  gc_ErrTranslation_en_Texts : ARRAY[0..1193] OF POINTER TO WSTRING(101) := [ADR(gc_ErrTranslation_en_Text0), ADR(gc_ErrTranslation_en_Text1), ADR(gc_ErrTranslation_en_Text2), ADR(gc_ErrTranslation_en_Text3), ADR(gc_ErrTranslation_en_Text4), ADR(gc_ErrTranslation_en_Text5), ADR(gc_ErrTranslation_en_Text6), ADR(gc_ErrTranslation_en_Text7), ADR(gc_ErrTranslation_en_Text8), ADR(gc_ErrTranslation_en_Text9), ADR(gc_ErrTranslation_en_Text10), ADR(gc_ErrTranslation_en_Text11), ADR(gc_ErrTranslation_en_Text12), ADR(gc_ErrTranslation_en_Text13), ADR(gc_ErrTranslation_en_Text14), ADR(gc_ErrTranslation_en_Text15), ADR(gc_ErrTranslation_en_Text16), ADR(gc_ErrTranslation_en_Text17), ADR(gc_ErrTranslation_en_Text18), ADR(gc_ErrTranslation_en_Text19), ADR(gc_ErrTranslation_en_Text20), ADR(gc_ErrTranslation_en_Text21), ADR(gc_ErrTranslation_en_Text22), ADR(gc_ErrTranslation_en_Text23), ADR(gc_ErrTranslation_en_Text24), ADR(gc_ErrTranslation_en_Text25), ADR(gc_ErrTranslation_en_Text26), ADR(gc_ErrTranslation_en_Text27), ADR(gc_ErrTranslation_en_Text28), ADR(gc_ErrTranslation_en_Text29), ADR(gc_ErrTranslation_en_Text30), ADR(gc_ErrTranslation_en_Text31), ADR(gc_ErrTranslation_en_Text32), ADR(gc_ErrTranslation_en_Text33), ADR(gc_ErrTranslation_en_Text34), ADR(gc_ErrTranslation_en_Text35), ADR(gc_ErrTranslation_en_Text36), ADR(gc_ErrTranslation_en_Text37), ADR(gc_ErrTranslation_en_Text38), ADR(gc_ErrTranslation_en_Text39), ADR(gc_ErrTranslation_en_Text40), ADR(gc_ErrTranslation_en_Text41), ADR(gc_ErrTranslation_en_Text42), ADR(gc_ErrTranslation_en_Text43), ADR(gc_ErrTranslation_en_Text44), ADR(gc_ErrTranslation_en_Text45), ADR(gc_ErrTranslation_en_Text46), ADR(gc_ErrTranslation_en_Text47), ADR(gc_ErrTranslation_en_Text48), ADR(gc_ErrTranslation_en_Text49), ADR(gc_ErrTranslation_en_Text50), ADR(gc_ErrTranslation_en_Text51), ADR(gc_ErrTranslation_en_Text52), ADR(gc_ErrTranslation_en_Text53), ADR(gc_ErrTranslation_en_Text54), ADR(gc_ErrTranslation_en_Text55), ADR(gc_ErrTranslation_en_Text56), ADR(gc_ErrTranslation_en_Text57), ADR(gc_ErrTranslation_en_Text58), ADR(gc_ErrTranslation_en_Text59), ADR(gc_ErrTranslation_en_Text60), ADR(gc_ErrTranslation_en_Text61), ADR(gc_ErrTranslation_en_Text62), ADR(gc_ErrTranslation_en_Text63), ADR(gc_ErrTranslation_en_Text64), ADR(gc_ErrTranslation_en_Text65), ADR(gc_ErrTranslation_en_Text66), ADR(gc_ErrTranslation_en_Text67), ADR(gc_ErrTranslation_en_Text68), ADR(gc_ErrTranslation_en_Text69), ADR(gc_ErrTranslation_en_Text70), ADR(gc_ErrTranslation_en_Text71), ADR(gc_ErrTranslation_en_Text72), ADR(gc_ErrTranslation_en_Text73), ADR(gc_ErrTranslation_en_Text74), ADR(gc_ErrTranslation_en_Text75), ADR(gc_ErrTranslation_en_Text76), ADR(gc_ErrTranslation_en_Text77), ADR(gc_ErrTranslation_en_Text78), ADR(gc_ErrTranslation_en_Text79), ADR(gc_ErrTranslation_en_Text80), ADR(gc_ErrTranslation_en_Text81), ADR(gc_ErrTranslation_en_Text82), ADR(gc_ErrTranslation_en_Text83), ADR(gc_ErrTranslation_en_Text84), ADR(gc_ErrTranslation_en_Text85), ADR(gc_ErrTranslation_en_Text86), ADR(gc_ErrTranslation_en_Text87), ADR(gc_ErrTranslation_en_Text88), ADR(gc_ErrTranslation_en_Text89), ADR(gc_ErrTranslation_en_Text90), ADR(gc_ErrTranslation_en_Text91), ADR(gc_ErrTranslation_en_Text92), ADR(gc_ErrTranslation_en_Text93), ADR(gc_ErrTranslation_en_Text94), ADR(gc_ErrTranslation_en_Text95), ADR(gc_ErrTranslation_en_Text96), ADR(gc_ErrTranslation_en_Text97), ADR(gc_ErrTranslation_en_Text98), ADR(gc_ErrTranslation_en_Text99), ADR(gc_ErrTranslation_en_Text100), ADR(gc_ErrTranslation_en_Text101), ADR(gc_ErrTranslation_en_Text102), ADR(gc_ErrTranslation_en_Text103), ADR(gc_ErrTranslation_en_Text104), ADR(gc_ErrTranslation_en_Text105), ADR(gc_ErrTranslation_en_Text106), ADR(gc_ErrTranslation_en_Text107), ADR(gc_ErrTranslation_en_Text108), ADR(gc_ErrTranslation_en_Text109), ADR(gc_ErrTranslation_en_Text110), ADR(gc_ErrTranslation_en_Text111), ADR(gc_ErrTranslation_en_Text112), ADR(gc_ErrTranslation_en_Text113), ADR(gc_ErrTranslation_en_Text114), ADR(gc_ErrTranslation_en_Text115), ADR(gc_ErrTranslation_en_Text116), ADR(gc_ErrTranslation_en_Text117), ADR(gc_ErrTranslation_en_Text118), ADR(gc_ErrTranslation_en_Text119), ADR(gc_ErrTranslation_en_Text120), ADR(gc_ErrTranslation_en_Text121), ADR(gc_ErrTranslation_en_Text122), ADR(gc_ErrTranslation_en_Text123), ADR(gc_ErrTranslation_en_Text124), ADR(gc_ErrTranslation_en_Text125), ADR(gc_ErrTranslation_en_Text126), ADR(gc_ErrTranslation_en_Text127), ADR(gc_ErrTranslation_en_Text128), ADR(gc_ErrTranslation_en_Text129), ADR(gc_ErrTranslation_en_Text130), ADR(gc_ErrTranslation_en_Text131), ADR(gc_ErrTranslation_en_Text132), ADR(gc_ErrTranslation_en_Text133), ADR(gc_ErrTranslation_en_Text134), ADR(gc_ErrTranslation_en_Text135), ADR(gc_ErrTranslation_en_Text136), ADR(gc_ErrTranslation_en_Text137), ADR(gc_ErrTranslation_en_Text138), ADR(gc_ErrTranslation_en_Text139), ADR(gc_ErrTranslation_en_Text140), ADR(gc_ErrTranslation_en_Text141), ADR(gc_ErrTranslation_en_Text142), ADR(gc_ErrTranslation_en_Text143), ADR(gc_ErrTranslation_en_Text144), ADR(gc_ErrTranslation_en_Text145), ADR(gc_ErrTranslation_en_Text146), ADR(gc_ErrTranslation_en_Text147), ADR(gc_ErrTranslation_en_Text148), ADR(gc_ErrTranslation_en_Text149), ADR(gc_ErrTranslation_en_Text150), ADR(gc_ErrTranslation_en_Text151), ADR(gc_ErrTranslation_en_Text152), ADR(gc_ErrTranslation_en_Text153), ADR(gc_ErrTranslation_en_Text154), ADR(gc_ErrTranslation_en_Text155), ADR(gc_ErrTranslation_en_Text156), ADR(gc_ErrTranslation_en_Text157), ADR(gc_ErrTranslation_en_Text158), ADR(gc_ErrTranslation_en_Text159), ADR(gc_ErrTranslation_en_Text160), ADR(gc_ErrTranslation_en_Text161), ADR(gc_ErrTranslation_en_Text162), ADR(gc_ErrTranslation_en_Text163), ADR(gc_ErrTranslation_en_Text164), ADR(gc_ErrTranslation_en_Text165), ADR(gc_ErrTranslation_en_Text166), ADR(gc_ErrTranslation_en_Text167), ADR(gc_ErrTranslation_en_Text168), ADR(gc_ErrTranslation_en_Text169), ADR(gc_ErrTranslation_en_Text170), ADR(gc_ErrTranslation_en_Text171), ADR(gc_ErrTranslation_en_Text172), ADR(gc_ErrTranslation_en_Text173), ADR(gc_ErrTranslation_en_Text174), ADR(gc_ErrTranslation_en_Text175), ADR(gc_ErrTranslation_en_Text176), ADR(gc_ErrTranslation_en_Text177), ADR(gc_ErrTranslation_en_Text178), ADR(gc_ErrTranslation_en_Text179), ADR(gc_ErrTranslation_en_Text180), ADR(gc_ErrTranslation_en_Text181), ADR(gc_ErrTranslation_en_Text182), ADR(gc_ErrTranslation_en_Text183), ADR(gc_ErrTranslation_en_Text184), ADR(gc_ErrTranslation_en_Text185), ADR(gc_ErrTranslation_en_Text186), ADR(gc_ErrTranslation_en_Text187), ADR(gc_ErrTranslation_en_Text188), ADR(gc_ErrTranslation_en_Text189), ADR(gc_ErrTranslation_en_Text190), ADR(gc_ErrTranslation_en_Text191), ADR(gc_ErrTranslation_en_Text192), ADR(gc_ErrTranslation_en_Text193), ADR(gc_ErrTranslation_en_Text194), ADR(gc_ErrTranslation_en_Text195), ADR(gc_ErrTranslation_en_Text196), ADR(gc_ErrTranslation_en_Text197), ADR(gc_ErrTranslation_en_Text198), ADR(gc_ErrTranslation_en_Text199), ADR(gc_ErrTranslation_en_Text200), ADR(gc_ErrTranslation_en_Text201), ADR(gc_ErrTranslation_en_Text202), ADR(gc_ErrTranslation_en_Text203), ADR(gc_ErrTranslation_en_Text204), ADR(gc_ErrTranslation_en_Text205), ADR(gc_ErrTranslation_en_Text206), ADR(gc_ErrTranslation_en_Text207), ADR(gc_ErrTranslation_en_Text208), ADR(gc_ErrTranslation_en_Text209), ADR(gc_ErrTranslation_en_Text210), ADR(gc_ErrTranslation_en_Text211), ADR(gc_ErrTranslation_en_Text212), ADR(gc_ErrTranslation_en_Text213), ADR(gc_ErrTranslation_en_Text214), ADR(gc_ErrTranslation_en_Text215), ADR(gc_ErrTranslation_en_Text216), ADR(gc_ErrTranslation_en_Text217), ADR(gc_ErrTranslation_en_Text218), ADR(gc_ErrTranslation_en_Text219), ADR(gc_ErrTranslation_en_Text220), ADR(gc_ErrTranslation_en_Text221), ADR(gc_ErrTranslation_en_Text222), ADR(gc_ErrTranslation_en_Text223), ADR(gc_ErrTranslation_en_Text224), ADR(gc_ErrTranslation_en_Text225), ADR(gc_ErrTranslation_en_Text226), ADR(gc_ErrTranslation_en_Text227), ADR(gc_ErrTranslation_en_Text228), ADR(gc_ErrTranslation_en_Text229), ADR(gc_ErrTranslation_en_Text230), ADR(gc_ErrTranslation_en_Text231), ADR(gc_ErrTranslation_en_Text232), ADR(gc_ErrTranslation_en_Text233), ADR(gc_ErrTranslation_en_Text234), ADR(gc_ErrTranslation_en_Text235), ADR(gc_ErrTranslation_en_Text236), ADR(gc_ErrTranslation_en_Text237), ADR(gc_ErrTranslation_en_Text238), ADR(gc_ErrTranslation_en_Text239), ADR(gc_ErrTranslation_en_Text240), ADR(gc_ErrTranslation_en_Text241), ADR(gc_ErrTranslation_en_Text242), ADR(gc_ErrTranslation_en_Text243), ADR(gc_ErrTranslation_en_Text244), ADR(gc_ErrTranslation_en_Text245), ADR(gc_ErrTranslation_en_Text246), ADR(gc_ErrTranslation_en_Text247), ADR(gc_ErrTranslation_en_Text248), ADR(gc_ErrTranslation_en_Text249), ADR(gc_ErrTranslation_en_Text250), ADR(gc_ErrTranslation_en_Text251), ADR(gc_ErrTranslation_en_Text252), ADR(gc_ErrTranslation_en_Text253), ADR(gc_ErrTranslation_en_Text254), ADR(gc_ErrTranslation_en_Text255), ADR(gc_ErrTranslation_en_Text256), ADR(gc_ErrTranslation_en_Text257), ADR(gc_ErrTranslation_en_Text258), ADR(gc_ErrTranslation_en_Text259), ADR(gc_ErrTranslation_en_Text260), ADR(gc_ErrTranslation_en_Text261), ADR(gc_ErrTranslation_en_Text262), ADR(gc_ErrTranslation_en_Text263), ADR(gc_ErrTranslation_en_Text264), ADR(gc_ErrTranslation_en_Text265), ADR(gc_ErrTranslation_en_Text266), ADR(gc_ErrTranslation_en_Text267), ADR(gc_ErrTranslation_en_Text268), ADR(gc_ErrTranslation_en_Text269), ADR(gc_ErrTranslation_en_Text270), ADR(gc_ErrTranslation_en_Text271), ADR(gc_ErrTranslation_en_Text272), ADR(gc_ErrTranslation_en_Text273), ADR(gc_ErrTranslation_en_Text274), ADR(gc_ErrTranslation_en_Text275), ADR(gc_ErrTranslation_en_Text276), ADR(gc_ErrTranslation_en_Text277), ADR(gc_ErrTranslation_en_Text278), ADR(gc_ErrTranslation_en_Text279), ADR(gc_ErrTranslation_en_Text280), ADR(gc_ErrTranslation_en_Text281), ADR(gc_ErrTranslation_en_Text282), ADR(gc_ErrTranslation_en_Text283), ADR(gc_ErrTranslation_en_Text284), ADR(gc_ErrTranslation_en_Text285), ADR(gc_ErrTranslation_en_Text286), ADR(gc_ErrTranslation_en_Text287), ADR(gc_ErrTranslation_en_Text288), ADR(gc_ErrTranslation_en_Text289), ADR(gc_ErrTranslation_en_Text290), ADR(gc_ErrTranslation_en_Text291), ADR(gc_ErrTranslation_en_Text292), ADR(gc_ErrTranslation_en_Text293), ADR(gc_ErrTranslation_en_Text294), ADR(gc_ErrTranslation_en_Text295), ADR(gc_ErrTranslation_en_Text296), ADR(gc_ErrTranslation_en_Text297), ADR(gc_ErrTranslation_en_Text298), ADR(gc_ErrTranslation_en_Text299), ADR(gc_ErrTranslation_en_Text300), ADR(gc_ErrTranslation_en_Text301), ADR(gc_ErrTranslation_en_Text302), ADR(gc_ErrTranslation_en_Text303), ADR(gc_ErrTranslation_en_Text304), ADR(gc_ErrTranslation_en_Text305), ADR(gc_ErrTranslation_en_Text306), ADR(gc_ErrTranslation_en_Text307), ADR(gc_ErrTranslation_en_Text308), ADR(gc_ErrTranslation_en_Text309), ADR(gc_ErrTranslation_en_Text310), ADR(gc_ErrTranslation_en_Text311), ADR(gc_ErrTranslation_en_Text312), ADR(gc_ErrTranslation_en_Text313), ADR(gc_ErrTranslation_en_Text314), ADR(gc_ErrTranslation_en_Text315), ADR(gc_ErrTranslation_en_Text316), ADR(gc_ErrTranslation_en_Text317), ADR(gc_ErrTranslation_en_Text318), ADR(gc_ErrTranslation_en_Text319), ADR(gc_ErrTranslation_en_Text320), ADR(gc_ErrTranslation_en_Text321), ADR(gc_ErrTranslation_en_Text322), ADR(gc_ErrTranslation_en_Text323), ADR(gc_ErrTranslation_en_Text324), ADR(gc_ErrTranslation_en_Text325), ADR(gc_ErrTranslation_en_Text326), ADR(gc_ErrTranslation_en_Text327), ADR(gc_ErrTranslation_en_Text328), ADR(gc_ErrTranslation_en_Text329), ADR(gc_ErrTranslation_en_Text330), ADR(gc_ErrTranslation_en_Text331), ADR(gc_ErrTranslation_en_Text332), ADR(gc_ErrTranslation_en_Text333), ADR(gc_ErrTranslation_en_Text334), ADR(gc_ErrTranslation_en_Text335), ADR(gc_ErrTranslation_en_Text336), ADR(gc_ErrTranslation_en_Text337), ADR(gc_ErrTranslation_en_Text338), ADR(gc_ErrTranslation_en_Text339), ADR(gc_ErrTranslation_en_Text340), ADR(gc_ErrTranslation_en_Text341), ADR(gc_ErrTranslation_en_Text342), ADR(gc_ErrTranslation_en_Text343), ADR(gc_ErrTranslation_en_Text344), ADR(gc_ErrTranslation_en_Text345), ADR(gc_ErrTranslation_en_Text346), ADR(gc_ErrTranslation_en_Text347), ADR(gc_ErrTranslation_en_Text348), ADR(gc_ErrTranslation_en_Text349), ADR(gc_ErrTranslation_en_Text350), ADR(gc_ErrTranslation_en_Text351), ADR(gc_ErrTranslation_en_Text352), ADR(gc_ErrTranslation_en_Text353), ADR(gc_ErrTranslation_en_Text354), ADR(gc_ErrTranslation_en_Text355), ADR(gc_ErrTranslation_en_Text356), ADR(gc_ErrTranslation_en_Text357), ADR(gc_ErrTranslation_en_Text358), ADR(gc_ErrTranslation_en_Text359), ADR(gc_ErrTranslation_en_Text360), ADR(gc_ErrTranslation_en_Text361), ADR(gc_ErrTranslation_en_Text362), ADR(gc_ErrTranslation_en_Text363), ADR(gc_ErrTranslation_en_Text364), ADR(gc_ErrTranslation_en_Text365), ADR(gc_ErrTranslation_en_Text366), ADR(gc_ErrTranslation_en_Text367), ADR(gc_ErrTranslation_en_Text368), ADR(gc_ErrTranslation_en_Text369), ADR(gc_ErrTranslation_en_Text370), ADR(gc_ErrTranslation_en_Text371), ADR(gc_ErrTranslation_en_Text372), ADR(gc_ErrTranslation_en_Text373), ADR(gc_ErrTranslation_en_Text374), ADR(gc_ErrTranslation_en_Text375), ADR(gc_ErrTranslation_en_Text376), ADR(gc_ErrTranslation_en_Text377), ADR(gc_ErrTranslation_en_Text378), ADR(gc_ErrTranslation_en_Text379), ADR(gc_ErrTranslation_en_Text380), ADR(gc_ErrTranslation_en_Text381), ADR(gc_ErrTranslation_en_Text382), ADR(gc_ErrTranslation_en_Text383), ADR(gc_ErrTranslation_en_Text384), ADR(gc_ErrTranslation_en_Text385), ADR(gc_ErrTranslation_en_Text386), ADR(gc_ErrTranslation_en_Text387), ADR(gc_ErrTranslation_en_Text388), ADR(gc_ErrTranslation_en_Text389), ADR(gc_ErrTranslation_en_Text390), ADR(gc_ErrTranslation_en_Text391), ADR(gc_ErrTranslation_en_Text392), ADR(gc_ErrTranslation_en_Text393), ADR(gc_ErrTranslation_en_Text394), ADR(gc_ErrTranslation_en_Text395), ADR(gc_ErrTranslation_en_Text396), ADR(gc_ErrTranslation_en_Text397), ADR(gc_ErrTranslation_en_Text398), ADR(gc_ErrTranslation_en_Text399), ADR(gc_ErrTranslation_en_Text400), ADR(gc_ErrTranslation_en_Text401), ADR(gc_ErrTranslation_en_Text402), ADR(gc_ErrTranslation_en_Text403), ADR(gc_ErrTranslation_en_Text404), ADR(gc_ErrTranslation_en_Text405), ADR(gc_ErrTranslation_en_Text406), ADR(gc_ErrTranslation_en_Text407), ADR(gc_ErrTranslation_en_Text408), ADR(gc_ErrTranslation_en_Text409), ADR(gc_ErrTranslation_en_Text410), ADR(gc_ErrTranslation_en_Text411), ADR(gc_ErrTranslation_en_Text412), ADR(gc_ErrTranslation_en_Text413), ADR(gc_ErrTranslation_en_Text414), ADR(gc_ErrTranslation_en_Text415), ADR(gc_ErrTranslation_en_Text416), ADR(gc_ErrTranslation_en_Text417), ADR(gc_ErrTranslation_en_Text418), ADR(gc_ErrTranslation_en_Text419), ADR(gc_ErrTranslation_en_Text420), ADR(gc_ErrTranslation_en_Text421), ADR(gc_ErrTranslation_en_Text422), ADR(gc_ErrTranslation_en_Text423), ADR(gc_ErrTranslation_en_Text424), ADR(gc_ErrTranslation_en_Text425), ADR(gc_ErrTranslation_en_Text426), ADR(gc_ErrTranslation_en_Text427), ADR(gc_ErrTranslation_en_Text428), ADR(gc_ErrTranslation_en_Text429), ADR(gc_ErrTranslation_en_Text430), ADR(gc_ErrTranslation_en_Text431), ADR(gc_ErrTranslation_en_Text432), ADR(gc_ErrTranslation_en_Text433), ADR(gc_ErrTranslation_en_Text434), ADR(gc_ErrTranslation_en_Text435), ADR(gc_ErrTranslation_en_Text436), ADR(gc_ErrTranslation_en_Text437), ADR(gc_ErrTranslation_en_Text438), ADR(gc_ErrTranslation_en_Text439), ADR(gc_ErrTranslation_en_Text440), ADR(gc_ErrTranslation_en_Text441), ADR(gc_ErrTranslation_en_Text442), ADR(gc_ErrTranslation_en_Text443), ADR(gc_ErrTranslation_en_Text444), ADR(gc_ErrTranslation_en_Text445), ADR(gc_ErrTranslation_en_Text446), ADR(gc_ErrTranslation_en_Text447), ADR(gc_ErrTranslation_en_Text448), ADR(gc_ErrTranslation_en_Text449), ADR(gc_ErrTranslation_en_Text450), ADR(gc_ErrTranslation_en_Text451), ADR(gc_ErrTranslation_en_Text452), ADR(gc_ErrTranslation_en_Text453), ADR(gc_ErrTranslation_en_Text454), ADR(gc_ErrTranslation_en_Text455), ADR(gc_ErrTranslation_en_Text456), ADR(gc_ErrTranslation_en_Text457), ADR(gc_ErrTranslation_en_Text458), ADR(gc_ErrTranslation_en_Text459), ADR(gc_ErrTranslation_en_Text460), ADR(gc_ErrTranslation_en_Text461), ADR(gc_ErrTranslation_en_Text462), ADR(gc_ErrTranslation_en_Text463), ADR(gc_ErrTranslation_en_Text464), ADR(gc_ErrTranslation_en_Text465), ADR(gc_ErrTranslation_en_Text466), ADR(gc_ErrTranslation_en_Text467), ADR(gc_ErrTranslation_en_Text468), ADR(gc_ErrTranslation_en_Text469), ADR(gc_ErrTranslation_en_Text470), ADR(gc_ErrTranslation_en_Text471), ADR(gc_ErrTranslation_en_Text472), ADR(gc_ErrTranslation_en_Text473), ADR(gc_ErrTranslation_en_Text474), ADR(gc_ErrTranslation_en_Text475), ADR(gc_ErrTranslation_en_Text476), ADR(gc_ErrTranslation_en_Text477), ADR(gc_ErrTranslation_en_Text478), ADR(gc_ErrTranslation_en_Text479), ADR(gc_ErrTranslation_en_Text480), ADR(gc_ErrTranslation_en_Text481), ADR(gc_ErrTranslation_en_Text482), ADR(gc_ErrTranslation_en_Text483), ADR(gc_ErrTranslation_en_Text484), ADR(gc_ErrTranslation_en_Text485), ADR(gc_ErrTranslation_en_Text486), ADR(gc_ErrTranslation_en_Text487), ADR(gc_ErrTranslation_en_Text488), ADR(gc_ErrTranslation_en_Text489), ADR(gc_ErrTranslation_en_Text490), ADR(gc_ErrTranslation_en_Text491), ADR(gc_ErrTranslation_en_Text492), ADR(gc_ErrTranslation_en_Text493), ADR(gc_ErrTranslation_en_Text494), ADR(gc_ErrTranslation_en_Text495), ADR(gc_ErrTranslation_en_Text496), ADR(gc_ErrTranslation_en_Text497), ADR(gc_ErrTranslation_en_Text498), ADR(gc_ErrTranslation_en_Text499), ADR(gc_ErrTranslation_en_Text500), ADR(gc_ErrTranslation_en_Text501), ADR(gc_ErrTranslation_en_Text502), ADR(gc_ErrTranslation_en_Text503), ADR(gc_ErrTranslation_en_Text504), ADR(gc_ErrTranslation_en_Text505), ADR(gc_ErrTranslation_en_Text506), ADR(gc_ErrTranslation_en_Text507), ADR(gc_ErrTranslation_en_Text508), ADR(gc_ErrTranslation_en_Text509), ADR(gc_ErrTranslation_en_Text510), ADR(gc_ErrTranslation_en_Text511), ADR(gc_ErrTranslation_en_Text512), ADR(gc_ErrTranslation_en_Text513), ADR(gc_ErrTranslation_en_Text514), ADR(gc_ErrTranslation_en_Text515), ADR(gc_ErrTranslation_en_Text516), ADR(gc_ErrTranslation_en_Text517), ADR(gc_ErrTranslation_en_Text518), ADR(gc_ErrTranslation_en_Text519), ADR(gc_ErrTranslation_en_Text520), ADR(gc_ErrTranslation_en_Text521), ADR(gc_ErrTranslation_en_Text522), ADR(gc_ErrTranslation_en_Text523), ADR(gc_ErrTranslation_en_Text524), ADR(gc_ErrTranslation_en_Text525), ADR(gc_ErrTranslation_en_Text526), ADR(gc_ErrTranslation_en_Text527), ADR(gc_ErrTranslation_en_Text528), ADR(gc_ErrTranslation_en_Text529), ADR(gc_ErrTranslation_en_Text530), ADR(gc_ErrTranslation_en_Text531), ADR(gc_ErrTranslation_en_Text532), ADR(gc_ErrTranslation_en_Text533), ADR(gc_ErrTranslation_en_Text534), ADR(gc_ErrTranslation_en_Text535), ADR(gc_ErrTranslation_en_Text536), ADR(gc_ErrTranslation_en_Text537), ADR(gc_ErrTranslation_en_Text538), ADR(gc_ErrTranslation_en_Text539), ADR(gc_ErrTranslation_en_Text540), ADR(gc_ErrTranslation_en_Text541), ADR(gc_ErrTranslation_en_Text542), ADR(gc_ErrTranslation_en_Text543), ADR(gc_ErrTranslation_en_Text544), ADR(gc_ErrTranslation_en_Text545), ADR(gc_ErrTranslation_en_Text546), ADR(gc_ErrTranslation_en_Text547), ADR(gc_ErrTranslation_en_Text548), ADR(gc_ErrTranslation_en_Text549), ADR(gc_ErrTranslation_en_Text550), ADR(gc_ErrTranslation_en_Text551), ADR(gc_ErrTranslation_en_Text552), ADR(gc_ErrTranslation_en_Text553), ADR(gc_ErrTranslation_en_Text554), ADR(gc_ErrTranslation_en_Text555), ADR(gc_ErrTranslation_en_Text556), ADR(gc_ErrTranslation_en_Text557), ADR(gc_ErrTranslation_en_Text558), ADR(gc_ErrTranslation_en_Text559), ADR(gc_ErrTranslation_en_Text560), ADR(gc_ErrTranslation_en_Text561), ADR(gc_ErrTranslation_en_Text562), ADR(gc_ErrTranslation_en_Text563), ADR(gc_ErrTranslation_en_Text564), ADR(gc_ErrTranslation_en_Text565), ADR(gc_ErrTranslation_en_Text566), ADR(gc_ErrTranslation_en_Text567), ADR(gc_ErrTranslation_en_Text568), ADR(gc_ErrTranslation_en_Text569), ADR(gc_ErrTranslation_en_Text570), ADR(gc_ErrTranslation_en_Text571), ADR(gc_ErrTranslation_en_Text572), ADR(gc_ErrTranslation_en_Text573), ADR(gc_ErrTranslation_en_Text574), ADR(gc_ErrTranslation_en_Text575), ADR(gc_ErrTranslation_en_Text576), ADR(gc_ErrTranslation_en_Text577), ADR(gc_ErrTranslation_en_Text578), ADR(gc_ErrTranslation_en_Text579), ADR(gc_ErrTranslation_en_Text580), ADR(gc_ErrTranslation_en_Text581), ADR(gc_ErrTranslation_en_Text582), ADR(gc_ErrTranslation_en_Text583), ADR(gc_ErrTranslation_en_Text584), ADR(gc_ErrTranslation_en_Text585), ADR(gc_ErrTranslation_en_Text586), ADR(gc_ErrTranslation_en_Text587), ADR(gc_ErrTranslation_en_Text588), ADR(gc_ErrTranslation_en_Text589), ADR(gc_ErrTranslation_en_Text590), ADR(gc_ErrTranslation_en_Text591), ADR(gc_ErrTranslation_en_Text592), ADR(gc_ErrTranslation_en_Text593), ADR(gc_ErrTranslation_en_Text594), ADR(gc_ErrTranslation_en_Text595), ADR(gc_ErrTranslation_en_Text596), ADR(gc_ErrTranslation_en_Text597), ADR(gc_ErrTranslation_en_Text598), ADR(gc_ErrTranslation_en_Text599), ADR(gc_ErrTranslation_en_Text600), ADR(gc_ErrTranslation_en_Text601), ADR(gc_ErrTranslation_en_Text602), ADR(gc_ErrTranslation_en_Text603), ADR(gc_ErrTranslation_en_Text604), ADR(gc_ErrTranslation_en_Text605), ADR(gc_ErrTranslation_en_Text606), ADR(gc_ErrTranslation_en_Text607), ADR(gc_ErrTranslation_en_Text608), ADR(gc_ErrTranslation_en_Text609), ADR(gc_ErrTranslation_en_Text610), ADR(gc_ErrTranslation_en_Text611), ADR(gc_ErrTranslation_en_Text612), ADR(gc_ErrTranslation_en_Text613), ADR(gc_ErrTranslation_en_Text614), ADR(gc_ErrTranslation_en_Text615), ADR(gc_ErrTranslation_en_Text616), ADR(gc_ErrTranslation_en_Text617), ADR(gc_ErrTranslation_en_Text618), ADR(gc_ErrTranslation_en_Text619), ADR(gc_ErrTranslation_en_Text620), ADR(gc_ErrTranslation_en_Text621), ADR(gc_ErrTranslation_en_Text622), ADR(gc_ErrTranslation_en_Text623), ADR(gc_ErrTranslation_en_Text624), ADR(gc_ErrTranslation_en_Text625), ADR(gc_ErrTranslation_en_Text626), ADR(gc_ErrTranslation_en_Text627), ADR(gc_ErrTranslation_en_Text628), ADR(gc_ErrTranslation_en_Text629), ADR(gc_ErrTranslation_en_Text630), ADR(gc_ErrTranslation_en_Text631), ADR(gc_ErrTranslation_en_Text632), ADR(gc_ErrTranslation_en_Text633), ADR(gc_ErrTranslation_en_Text634), ADR(gc_ErrTranslation_en_Text635), ADR(gc_ErrTranslation_en_Text636), ADR(gc_ErrTranslation_en_Text637), ADR(gc_ErrTranslation_en_Text638), ADR(gc_ErrTranslation_en_Text639), ADR(gc_ErrTranslation_en_Text640), ADR(gc_ErrTranslation_en_Text641), ADR(gc_ErrTranslation_en_Text642), ADR(gc_ErrTranslation_en_Text643), ADR(gc_ErrTranslation_en_Text644), ADR(gc_ErrTranslation_en_Text645), ADR(gc_ErrTranslation_en_Text646), ADR(gc_ErrTranslation_en_Text647), ADR(gc_ErrTranslation_en_Text648), ADR(gc_ErrTranslation_en_Text649), ADR(gc_ErrTranslation_en_Text650), ADR(gc_ErrTranslation_en_Text651), ADR(gc_ErrTranslation_en_Text652), ADR(gc_ErrTranslation_en_Text653), ADR(gc_ErrTranslation_en_Text654), ADR(gc_ErrTranslation_en_Text655), ADR(gc_ErrTranslation_en_Text656), ADR(gc_ErrTranslation_en_Text657), ADR(gc_ErrTranslation_en_Text658), ADR(gc_ErrTranslation_en_Text659), ADR(gc_ErrTranslation_en_Text660), ADR(gc_ErrTranslation_en_Text661), ADR(gc_ErrTranslation_en_Text662), ADR(gc_ErrTranslation_en_Text663), ADR(gc_ErrTranslation_en_Text664), ADR(gc_ErrTranslation_en_Text665), ADR(gc_ErrTranslation_en_Text666), ADR(gc_ErrTranslation_en_Text667), ADR(gc_ErrTranslation_en_Text668), ADR(gc_ErrTranslation_en_Text669), ADR(gc_ErrTranslation_en_Text670), ADR(gc_ErrTranslation_en_Text671), ADR(gc_ErrTranslation_en_Text672), ADR(gc_ErrTranslation_en_Text673), ADR(gc_ErrTranslation_en_Text674), ADR(gc_ErrTranslation_en_Text675), ADR(gc_ErrTranslation_en_Text676), ADR(gc_ErrTranslation_en_Text677), ADR(gc_ErrTranslation_en_Text678), ADR(gc_ErrTranslation_en_Text679), ADR(gc_ErrTranslation_en_Text680), ADR(gc_ErrTranslation_en_Text681), ADR(gc_ErrTranslation_en_Text682), ADR(gc_ErrTranslation_en_Text683), ADR(gc_ErrTranslation_en_Text684), ADR(gc_ErrTranslation_en_Text685), ADR(gc_ErrTranslation_en_Text686), ADR(gc_ErrTranslation_en_Text687), ADR(gc_ErrTranslation_en_Text688), ADR(gc_ErrTranslation_en_Text689), ADR(gc_ErrTranslation_en_Text690), ADR(gc_ErrTranslation_en_Text691), ADR(gc_ErrTranslation_en_Text692), ADR(gc_ErrTranslation_en_Text693), ADR(gc_ErrTranslation_en_Text694), ADR(gc_ErrTranslation_en_Text695), ADR(gc_ErrTranslation_en_Text696), ADR(gc_ErrTranslation_en_Text697), ADR(gc_ErrTranslation_en_Text698), ADR(gc_ErrTranslation_en_Text699), ADR(gc_ErrTranslation_en_Text700), ADR(gc_ErrTranslation_en_Text701), ADR(gc_ErrTranslation_en_Text702), ADR(gc_ErrTranslation_en_Text703), ADR(gc_ErrTranslation_en_Text704), ADR(gc_ErrTranslation_en_Text705), ADR(gc_ErrTranslation_en_Text706), ADR(gc_ErrTranslation_en_Text707), ADR(gc_ErrTranslation_en_Text708), ADR(gc_ErrTranslation_en_Text709), ADR(gc_ErrTranslation_en_Text710), ADR(gc_ErrTranslation_en_Text711), ADR(gc_ErrTranslation_en_Text712), ADR(gc_ErrTranslation_en_Text713), ADR(gc_ErrTranslation_en_Text714), ADR(gc_ErrTranslation_en_Text715), ADR(gc_ErrTranslation_en_Text716), ADR(gc_ErrTranslation_en_Text717), ADR(gc_ErrTranslation_en_Text718), ADR(gc_ErrTranslation_en_Text719), ADR(gc_ErrTranslation_en_Text720), ADR(gc_ErrTranslation_en_Text721), ADR(gc_ErrTranslation_en_Text722), ADR(gc_ErrTranslation_en_Text723), ADR(gc_ErrTranslation_en_Text724), ADR(gc_ErrTranslation_en_Text725), ADR(gc_ErrTranslation_en_Text726), ADR(gc_ErrTranslation_en_Text727), ADR(gc_ErrTranslation_en_Text728), ADR(gc_ErrTranslation_en_Text729), ADR(gc_ErrTranslation_en_Text730), ADR(gc_ErrTranslation_en_Text731), ADR(gc_ErrTranslation_en_Text732), ADR(gc_ErrTranslation_en_Text733), ADR(gc_ErrTranslation_en_Text734), ADR(gc_ErrTranslation_en_Text735), ADR(gc_ErrTranslation_en_Text736), ADR(gc_ErrTranslation_en_Text737), ADR(gc_ErrTranslation_en_Text738), ADR(gc_ErrTranslation_en_Text739), ADR(gc_ErrTranslation_en_Text740), ADR(gc_ErrTranslation_en_Text741), ADR(gc_ErrTranslation_en_Text742), ADR(gc_ErrTranslation_en_Text743), ADR(gc_ErrTranslation_en_Text744), ADR(gc_ErrTranslation_en_Text745), ADR(gc_ErrTranslation_en_Text746), ADR(gc_ErrTranslation_en_Text747), ADR(gc_ErrTranslation_en_Text748), ADR(gc_ErrTranslation_en_Text749), ADR(gc_ErrTranslation_en_Text750), ADR(gc_ErrTranslation_en_Text751), ADR(gc_ErrTranslation_en_Text752), ADR(gc_ErrTranslation_en_Text753), ADR(gc_ErrTranslation_en_Text754), ADR(gc_ErrTranslation_en_Text755), ADR(gc_ErrTranslation_en_Text756), ADR(gc_ErrTranslation_en_Text757), ADR(gc_ErrTranslation_en_Text758), ADR(gc_ErrTranslation_en_Text759), ADR(gc_ErrTranslation_en_Text760), ADR(gc_ErrTranslation_en_Text761), ADR(gc_ErrTranslation_en_Text762), ADR(gc_ErrTranslation_en_Text763), ADR(gc_ErrTranslation_en_Text764), ADR(gc_ErrTranslation_en_Text765), ADR(gc_ErrTranslation_en_Text766), ADR(gc_ErrTranslation_en_Text767), ADR(gc_ErrTranslation_en_Text768), ADR(gc_ErrTranslation_en_Text769), ADR(gc_ErrTranslation_en_Text770), ADR(gc_ErrTranslation_en_Text771), ADR(gc_ErrTranslation_en_Text772), ADR(gc_ErrTranslation_en_Text773), ADR(gc_ErrTranslation_en_Text774), ADR(gc_ErrTranslation_en_Text775), ADR(gc_ErrTranslation_en_Text776), ADR(gc_ErrTranslation_en_Text777), ADR(gc_ErrTranslation_en_Text778), ADR(gc_ErrTranslation_en_Text779), ADR(gc_ErrTranslation_en_Text780), ADR(gc_ErrTranslation_en_Text781), ADR(gc_ErrTranslation_en_Text782), ADR(gc_ErrTranslation_en_Text783), ADR(gc_ErrTranslation_en_Text784), ADR(gc_ErrTranslation_en_Text785), ADR(gc_ErrTranslation_en_Text786), ADR(gc_ErrTranslation_en_Text787), ADR(gc_ErrTranslation_en_Text788), ADR(gc_ErrTranslation_en_Text789), ADR(gc_ErrTranslation_en_Text790), ADR(gc_ErrTranslation_en_Text791), ADR(gc_ErrTranslation_en_Text792), ADR(gc_ErrTranslation_en_Text793), ADR(gc_ErrTranslation_en_Text794), ADR(gc_ErrTranslation_en_Text795), ADR(gc_ErrTranslation_en_Text796), ADR(gc_ErrTranslation_en_Text797), ADR(gc_ErrTranslation_en_Text798), ADR(gc_ErrTranslation_en_Text799), ADR(gc_ErrTranslation_en_Text800), ADR(gc_ErrTranslation_en_Text801), ADR(gc_ErrTranslation_en_Text802), ADR(gc_ErrTranslation_en_Text803), ADR(gc_ErrTranslation_en_Text804), ADR(gc_ErrTranslation_en_Text805), ADR(gc_ErrTranslation_en_Text806), ADR(gc_ErrTranslation_en_Text807), ADR(gc_ErrTranslation_en_Text808), ADR(gc_ErrTranslation_en_Text809), ADR(gc_ErrTranslation_en_Text810), ADR(gc_ErrTranslation_en_Text811), ADR(gc_ErrTranslation_en_Text812), ADR(gc_ErrTranslation_en_Text813), ADR(gc_ErrTranslation_en_Text814), ADR(gc_ErrTranslation_en_Text815), ADR(gc_ErrTranslation_en_Text816), ADR(gc_ErrTranslation_en_Text817), ADR(gc_ErrTranslation_en_Text818), ADR(gc_ErrTranslation_en_Text819), ADR(gc_ErrTranslation_en_Text820), ADR(gc_ErrTranslation_en_Text821), ADR(gc_ErrTranslation_en_Text822), ADR(gc_ErrTranslation_en_Text823), ADR(gc_ErrTranslation_en_Text824), ADR(gc_ErrTranslation_en_Text825), ADR(gc_ErrTranslation_en_Text826), ADR(gc_ErrTranslation_en_Text827), ADR(gc_ErrTranslation_en_Text828), ADR(gc_ErrTranslation_en_Text829), ADR(gc_ErrTranslation_en_Text830), ADR(gc_ErrTranslation_en_Text831), ADR(gc_ErrTranslation_en_Text832), ADR(gc_ErrTranslation_en_Text833), ADR(gc_ErrTranslation_en_Text834), ADR(gc_ErrTranslation_en_Text835), ADR(gc_ErrTranslation_en_Text836), ADR(gc_ErrTranslation_en_Text837), ADR(gc_ErrTranslation_en_Text838), ADR(gc_ErrTranslation_en_Text839), ADR(gc_ErrTranslation_en_Text840), ADR(gc_ErrTranslation_en_Text841), ADR(gc_ErrTranslation_en_Text842), ADR(gc_ErrTranslation_en_Text843), ADR(gc_ErrTranslation_en_Text844), ADR(gc_ErrTranslation_en_Text845), ADR(gc_ErrTranslation_en_Text846), ADR(gc_ErrTranslation_en_Text847), ADR(gc_ErrTranslation_en_Text848), ADR(gc_ErrTranslation_en_Text849), ADR(gc_ErrTranslation_en_Text850), ADR(gc_ErrTranslation_en_Text851), ADR(gc_ErrTranslation_en_Text852), ADR(gc_ErrTranslation_en_Text853), ADR(gc_ErrTranslation_en_Text854), ADR(gc_ErrTranslation_en_Text855), ADR(gc_ErrTranslation_en_Text856), ADR(gc_ErrTranslation_en_Text857), ADR(gc_ErrTranslation_en_Text858), ADR(gc_ErrTranslation_en_Text859), ADR(gc_ErrTranslation_en_Text860), ADR(gc_ErrTranslation_en_Text861), ADR(gc_ErrTranslation_en_Text862), ADR(gc_ErrTranslation_en_Text863), ADR(gc_ErrTranslation_en_Text864), ADR(gc_ErrTranslation_en_Text865), ADR(gc_ErrTranslation_en_Text866), ADR(gc_ErrTranslation_en_Text867), ADR(gc_ErrTranslation_en_Text868), ADR(gc_ErrTranslation_en_Text869), ADR(gc_ErrTranslation_en_Text870), ADR(gc_ErrTranslation_en_Text871), ADR(gc_ErrTranslation_en_Text872), ADR(gc_ErrTranslation_en_Text873), ADR(gc_ErrTranslation_en_Text874), ADR(gc_ErrTranslation_en_Text875), ADR(gc_ErrTranslation_en_Text876), ADR(gc_ErrTranslation_en_Text877), ADR(gc_ErrTranslation_en_Text878), ADR(gc_ErrTranslation_en_Text879), ADR(gc_ErrTranslation_en_Text880), ADR(gc_ErrTranslation_en_Text881), ADR(gc_ErrTranslation_en_Text882), ADR(gc_ErrTranslation_en_Text883), ADR(gc_ErrTranslation_en_Text884), ADR(gc_ErrTranslation_en_Text885), ADR(gc_ErrTranslation_en_Text886), ADR(gc_ErrTranslation_en_Text887), ADR(gc_ErrTranslation_en_Text888), ADR(gc_ErrTranslation_en_Text889), ADR(gc_ErrTranslation_en_Text890), ADR(gc_ErrTranslation_en_Text891), ADR(gc_ErrTranslation_en_Text892), ADR(gc_ErrTranslation_en_Text893), ADR(gc_ErrTranslation_en_Text894), ADR(gc_ErrTranslation_en_Text895), ADR(gc_ErrTranslation_en_Text896), ADR(gc_ErrTranslation_en_Text897), ADR(gc_ErrTranslation_en_Text898), ADR(gc_ErrTranslation_en_Text899), ADR(gc_ErrTranslation_en_Text900), ADR(gc_ErrTranslation_en_Text901), ADR(gc_ErrTranslation_en_Text902), ADR(gc_ErrTranslation_en_Text903), ADR(gc_ErrTranslation_en_Text904), ADR(gc_ErrTranslation_en_Text905), ADR(gc_ErrTranslation_en_Text906), ADR(gc_ErrTranslation_en_Text907), ADR(gc_ErrTranslation_en_Text908), ADR(gc_ErrTranslation_en_Text909), ADR(gc_ErrTranslation_en_Text910), ADR(gc_ErrTranslation_en_Text911), ADR(gc_ErrTranslation_en_Text912), ADR(gc_ErrTranslation_en_Text913), ADR(gc_ErrTranslation_en_Text914), ADR(gc_ErrTranslation_en_Text915), ADR(gc_ErrTranslation_en_Text916), ADR(gc_ErrTranslation_en_Text917), ADR(gc_ErrTranslation_en_Text918), ADR(gc_ErrTranslation_en_Text919), ADR(gc_ErrTranslation_en_Text920), ADR(gc_ErrTranslation_en_Text921), ADR(gc_ErrTranslation_en_Text922), ADR(gc_ErrTranslation_en_Text923), ADR(gc_ErrTranslation_en_Text924), ADR(gc_ErrTranslation_en_Text925), ADR(gc_ErrTranslation_en_Text926), ADR(gc_ErrTranslation_en_Text927), ADR(gc_ErrTranslation_en_Text928), ADR(gc_ErrTranslation_en_Text929), ADR(gc_ErrTranslation_en_Text930), ADR(gc_ErrTranslation_en_Text931), ADR(gc_ErrTranslation_en_Text932), ADR(gc_ErrTranslation_en_Text933), ADR(gc_ErrTranslation_en_Text934), ADR(gc_ErrTranslation_en_Text935), ADR(gc_ErrTranslation_en_Text936), ADR(gc_ErrTranslation_en_Text937), ADR(gc_ErrTranslation_en_Text938), ADR(gc_ErrTranslation_en_Text939), ADR(gc_ErrTranslation_en_Text940), ADR(gc_ErrTranslation_en_Text941), ADR(gc_ErrTranslation_en_Text942), ADR(gc_ErrTranslation_en_Text943), ADR(gc_ErrTranslation_en_Text944), ADR(gc_ErrTranslation_en_Text945), ADR(gc_ErrTranslation_en_Text946), ADR(gc_ErrTranslation_en_Text947), ADR(gc_ErrTranslation_en_Text948), ADR(gc_ErrTranslation_en_Text949), ADR(gc_ErrTranslation_en_Text950), ADR(gc_ErrTranslation_en_Text951), ADR(gc_ErrTranslation_en_Text952), ADR(gc_ErrTranslation_en_Text953), ADR(gc_ErrTranslation_en_Text954), ADR(gc_ErrTranslation_en_Text955), ADR(gc_ErrTranslation_en_Text956), ADR(gc_ErrTranslation_en_Text957), ADR(gc_ErrTranslation_en_Text958), ADR(gc_ErrTranslation_en_Text959), ADR(gc_ErrTranslation_en_Text960), ADR(gc_ErrTranslation_en_Text961), ADR(gc_ErrTranslation_en_Text962), ADR(gc_ErrTranslation_en_Text963), ADR(gc_ErrTranslation_en_Text964), ADR(gc_ErrTranslation_en_Text965), ADR(gc_ErrTranslation_en_Text966), ADR(gc_ErrTranslation_en_Text967), ADR(gc_ErrTranslation_en_Text968), ADR(gc_ErrTranslation_en_Text969), ADR(gc_ErrTranslation_en_Text970), ADR(gc_ErrTranslation_en_Text971), ADR(gc_ErrTranslation_en_Text972), ADR(gc_ErrTranslation_en_Text973), ADR(gc_ErrTranslation_en_Text974), ADR(gc_ErrTranslation_en_Text975), ADR(gc_ErrTranslation_en_Text976), ADR(gc_ErrTranslation_en_Text977), ADR(gc_ErrTranslation_en_Text978), ADR(gc_ErrTranslation_en_Text979), ADR(gc_ErrTranslation_en_Text980), ADR(gc_ErrTranslation_en_Text981), ADR(gc_ErrTranslation_en_Text982), ADR(gc_ErrTranslation_en_Text983), ADR(gc_ErrTranslation_en_Text984), ADR(gc_ErrTranslation_en_Text985), ADR(gc_ErrTranslation_en_Text986), ADR(gc_ErrTranslation_en_Text987), ADR(gc_ErrTranslation_en_Text988), ADR(gc_ErrTranslation_en_Text989), ADR(gc_ErrTranslation_en_Text990), ADR(gc_ErrTranslation_en_Text991), ADR(gc_ErrTranslation_en_Text992), ADR(gc_ErrTranslation_en_Text993), ADR(gc_ErrTranslation_en_Text994), ADR(gc_ErrTranslation_en_Text995), ADR(gc_ErrTranslation_en_Text996), ADR(gc_ErrTranslation_en_Text997), ADR(gc_ErrTranslation_en_Text998), ADR(gc_ErrTranslation_en_Text999), ADR(gc_ErrTranslation_en_Text1000), ADR(gc_ErrTranslation_en_Text1001), ADR(gc_ErrTranslation_en_Text1002), ADR(gc_ErrTranslation_en_Text1003), ADR(gc_ErrTranslation_en_Text1004), ADR(gc_ErrTranslation_en_Text1005), ADR(gc_ErrTranslation_en_Text1006), ADR(gc_ErrTranslation_en_Text1007), ADR(gc_ErrTranslation_en_Text1008), ADR(gc_ErrTranslation_en_Text1009), ADR(gc_ErrTranslation_en_Text1010), ADR(gc_ErrTranslation_en_Text1011), ADR(gc_ErrTranslation_en_Text1012), ADR(gc_ErrTranslation_en_Text1013), ADR(gc_ErrTranslation_en_Text1014), ADR(gc_ErrTranslation_en_Text1015), ADR(gc_ErrTranslation_en_Text1016), ADR(gc_ErrTranslation_en_Text1017), ADR(gc_ErrTranslation_en_Text1018), ADR(gc_ErrTranslation_en_Text1019), ADR(gc_ErrTranslation_en_Text1020), ADR(gc_ErrTranslation_en_Text1021), ADR(gc_ErrTranslation_en_Text1022), ADR(gc_ErrTranslation_en_Text1023), ADR(gc_ErrTranslation_en_Text1024), ADR(gc_ErrTranslation_en_Text1025), ADR(gc_ErrTranslation_en_Text1026), ADR(gc_ErrTranslation_en_Text1027), ADR(gc_ErrTranslation_en_Text1028), ADR(gc_ErrTranslation_en_Text1029), ADR(gc_ErrTranslation_en_Text1030), ADR(gc_ErrTranslation_en_Text1031), ADR(gc_ErrTranslation_en_Text1032), ADR(gc_ErrTranslation_en_Text1033), ADR(gc_ErrTranslation_en_Text1034), ADR(gc_ErrTranslation_en_Text1035), ADR(gc_ErrTranslation_en_Text1036), ADR(gc_ErrTranslation_en_Text1037), ADR(gc_ErrTranslation_en_Text1038), ADR(gc_ErrTranslation_en_Text1039), ADR(gc_ErrTranslation_en_Text1040), ADR(gc_ErrTranslation_en_Text1041), ADR(gc_ErrTranslation_en_Text1042), ADR(gc_ErrTranslation_en_Text1043), ADR(gc_ErrTranslation_en_Text1044), ADR(gc_ErrTranslation_en_Text1045), ADR(gc_ErrTranslation_en_Text1046), ADR(gc_ErrTranslation_en_Text1047), ADR(gc_ErrTranslation_en_Text1048), ADR(gc_ErrTranslation_en_Text1049), ADR(gc_ErrTranslation_en_Text1050), ADR(gc_ErrTranslation_en_Text1051), ADR(gc_ErrTranslation_en_Text1052), ADR(gc_ErrTranslation_en_Text1053), ADR(gc_ErrTranslation_en_Text1054), ADR(gc_ErrTranslation_en_Text1055), ADR(gc_ErrTranslation_en_Text1056), ADR(gc_ErrTranslation_en_Text1057), ADR(gc_ErrTranslation_en_Text1058), ADR(gc_ErrTranslation_en_Text1059), ADR(gc_ErrTranslation_en_Text1060), ADR(gc_ErrTranslation_en_Text1061), ADR(gc_ErrTranslation_en_Text1062), ADR(gc_ErrTranslation_en_Text1063), ADR(gc_ErrTranslation_en_Text1064), ADR(gc_ErrTranslation_en_Text1065), ADR(gc_ErrTranslation_en_Text1066), ADR(gc_ErrTranslation_en_Text1067), ADR(gc_ErrTranslation_en_Text1068), ADR(gc_ErrTranslation_en_Text1069), ADR(gc_ErrTranslation_en_Text1070), ADR(gc_ErrTranslation_en_Text1071), ADR(gc_ErrTranslation_en_Text1072), ADR(gc_ErrTranslation_en_Text1073), ADR(gc_ErrTranslation_en_Text1074), ADR(gc_ErrTranslation_en_Text1075), ADR(gc_ErrTranslation_en_Text1076), ADR(gc_ErrTranslation_en_Text1077), ADR(gc_ErrTranslation_en_Text1078), ADR(gc_ErrTranslation_en_Text1079), ADR(gc_ErrTranslation_en_Text1080), ADR(gc_ErrTranslation_en_Text1081), ADR(gc_ErrTranslation_en_Text1082), ADR(gc_ErrTranslation_en_Text1083), ADR(gc_ErrTranslation_en_Text1084), ADR(gc_ErrTranslation_en_Text1085), ADR(gc_ErrTranslation_en_Text1086), ADR(gc_ErrTranslation_en_Text1087), ADR(gc_ErrTranslation_en_Text1088), ADR(gc_ErrTranslation_en_Text1089), ADR(gc_ErrTranslation_en_Text1090), ADR(gc_ErrTranslation_en_Text1091), ADR(gc_ErrTranslation_en_Text1092), ADR(gc_ErrTranslation_en_Text1093), ADR(gc_ErrTranslation_en_Text1094), ADR(gc_ErrTranslation_en_Text1095), ADR(gc_ErrTranslation_en_Text1096), ADR(gc_ErrTranslation_en_Text1097), ADR(gc_ErrTranslation_en_Text1098), ADR(gc_ErrTranslation_en_Text1099), ADR(gc_ErrTranslation_en_Text1100), ADR(gc_ErrTranslation_en_Text1101), ADR(gc_ErrTranslation_en_Text1102), ADR(gc_ErrTranslation_en_Text1103), ADR(gc_ErrTranslation_en_Text1104), ADR(gc_ErrTranslation_en_Text1105), ADR(gc_ErrTranslation_en_Text1106), ADR(gc_ErrTranslation_en_Text1107), ADR(gc_ErrTranslation_en_Text1108), ADR(gc_ErrTranslation_en_Text1109), ADR(gc_ErrTranslation_en_Text1110), ADR(gc_ErrTranslation_en_Text1111), ADR(gc_ErrTranslation_en_Text1112), ADR(gc_ErrTranslation_en_Text1113), ADR(gc_ErrTranslation_en_Text1114), ADR(gc_ErrTranslation_en_Text1115), ADR(gc_ErrTranslation_en_Text1116), ADR(gc_ErrTranslation_en_Text1117), ADR(gc_ErrTranslation_en_Text1118), ADR(gc_ErrTranslation_en_Text1119), ADR(gc_ErrTranslation_en_Text1120), ADR(gc_ErrTranslation_en_Text1121), ADR(gc_ErrTranslation_en_Text1122), ADR(gc_ErrTranslation_en_Text1123), ADR(gc_ErrTranslation_en_Text1124), ADR(gc_ErrTranslation_en_Text1125), ADR(gc_ErrTranslation_en_Text1126), ADR(gc_ErrTranslation_en_Text1127), ADR(gc_ErrTranslation_en_Text1128), ADR(gc_ErrTranslation_en_Text1129), ADR(gc_ErrTranslation_en_Text1130), ADR(gc_ErrTranslation_en_Text1131), ADR(gc_ErrTranslation_en_Text1132), ADR(gc_ErrTranslation_en_Text1133), ADR(gc_ErrTranslation_en_Text1134), ADR(gc_ErrTranslation_en_Text1135), ADR(gc_ErrTranslation_en_Text1136), ADR(gc_ErrTranslation_en_Text1137), ADR(gc_ErrTranslation_en_Text1138), ADR(gc_ErrTranslation_en_Text1139), ADR(gc_ErrTranslation_en_Text1140), ADR(gc_ErrTranslation_en_Text1141), ADR(gc_ErrTranslation_en_Text1142), ADR(gc_ErrTranslation_en_Text1143), ADR(gc_ErrTranslation_en_Text1144), ADR(gc_ErrTranslation_en_Text1145), ADR(gc_ErrTranslation_en_Text1146), ADR(gc_ErrTranslation_en_Text1147), ADR(gc_ErrTranslation_en_Text1148), ADR(gc_ErrTranslation_en_Text1149), ADR(gc_ErrTranslation_en_Text1150), ADR(gc_ErrTranslation_en_Text1151), ADR(gc_ErrTranslation_en_Text1152), ADR(gc_ErrTranslation_en_Text1153), ADR(gc_ErrTranslation_en_Text1154), ADR(gc_ErrTranslation_en_Text1155), ADR(gc_ErrTranslation_en_Text1156), ADR(gc_ErrTranslation_en_Text1157), ADR(gc_ErrTranslation_en_Text1158), ADR(gc_ErrTranslation_en_Text1159), ADR(gc_ErrTranslation_en_Text1160), ADR(gc_ErrTranslation_en_Text1161), ADR(gc_ErrTranslation_en_Text1162), ADR(gc_ErrTranslation_en_Text1163), ADR(gc_ErrTranslation_en_Text1164), ADR(gc_ErrTranslation_en_Text1165), ADR(gc_ErrTranslation_en_Text1166), ADR(gc_ErrTranslation_en_Text1167), ADR(gc_ErrTranslation_en_Text1168), ADR(gc_ErrTranslation_en_Text1169), ADR(gc_ErrTranslation_en_Text1170), ADR(gc_ErrTranslation_en_Text1171), ADR(gc_ErrTranslation_en_Text1172), ADR(gc_ErrTranslation_en_Text1173), ADR(gc_ErrTranslation_en_Text1174), ADR(gc_ErrTranslation_en_Text1175), ADR(gc_ErrTranslation_en_Text1176), ADR(gc_ErrTranslation_en_Text1177), ADR(gc_ErrTranslation_en_Text1178), ADR(gc_ErrTranslation_en_Text1179), ADR(gc_ErrTranslation_en_Text1180), ADR(gc_ErrTranslation_en_Text1181), ADR(gc_ErrTranslation_en_Text1182), ADR(gc_ErrTranslation_en_Text1183), ADR(gc_ErrTranslation_en_Text1184), ADR(gc_ErrTranslation_en_Text1185), ADR(gc_ErrTranslation_en_Text1186), ADR(gc_ErrTranslation_en_Text1187), ADR(gc_ErrTranslation_en_Text1188), ADR(gc_ErrTranslation_en_Text1189), ADR(gc_ErrTranslation_en_Text1190), ADR(gc_ErrTranslation_en_Text1191), ADR(gc_ErrTranslation_en_Text1192), ADR(gc_ErrTranslation_en_Text1193)];
  gc_ErrTranslation_en : TTranslation := (IsoCode := 'en', EnglishName := "english", NativeName := "english", Texts := ADR(gc_ErrTranslation_en_Texts));
  gc_ErrTranslation_fr_Text0 : WSTRING(40) := " [-]: Ecu0_Safety -  DM_ECU0_INPBOARDNON";
  gc_ErrTranslation_fr_Text1 : WSTRING(40) := " [-]: Ecu0_Safety -  DM_ECU0_INPBOARDFAT";
  gc_ErrTranslation_fr_Text2 : WSTRING(38) := " [-]: Ecu0_Safety -  DM_ECU0_INPUTPINS";
  gc_ErrTranslation_fr_Text3 : WSTRING(67) := " [-]: Ecu0_Safety -  Digital pin error - check ECU hardware and EMI";
  gc_ErrTranslation_fr_Text4 : WSTRING(66) := " [-]: Ecu0_Safety -  PWM output error - check ECU hardware and EMI";
  gc_ErrTranslation_fr_Text5 : WSTRING(63) := " [-]: Ecu0_Safety -  CPU core error - check source code and EMI";
  gc_ErrTranslation_fr_Text6 : WSTRING(33) := " [-]: Ecu0_Safety -  Memory error";
  gc_ErrTranslation_fr_Text7 : WSTRING(86) := " [-]: Ecu0_Safety -  Error during watchdog startup - check watchdog timing constraints";
  gc_ErrTranslation_fr_Text8 : WSTRING(88) := " [-]: Ecu1_Safety -  Safety switch error - check external shut-off pins and ECU hardware";
  gc_ErrTranslation_fr_Text9 : WSTRING(55) := " [-]: Ecu1_Safety -  Application code called safe state";
  gc_ErrTranslation_fr_Text10 : WSTRING(29) := " [-]: CAN_BUS0 -  CAN Bus off";
  gc_ErrTranslation_fr_Text11 : WSTRING(29) := " [-]: CAN_BUS0 -  CAN warning";
  gc_ErrTranslation_fr_Text12 : WSTRING(65) := " [-]: Ecu1_Safety -  Fatal error caused safe state -  replace ECU";
  gc_ErrTranslation_fr_Text13 : WSTRING(62) := " [-]: Ecu1_Safety -  BSP error caused safe state - replace ECU";
  gc_ErrTranslation_fr_Text14 : WSTRING(29) := " [-]: EcuSil -  Task overload";
  gc_ErrTranslation_fr_Text15 : WSTRING(28) := " [-]: EcuSil -  Batttery Low";
  gc_ErrTranslation_fr_Text16 : WSTRING(28) := " [-]: EcuSil -  Battery High";
  gc_ErrTranslation_fr_Text17 : WSTRING(31) := " [-]: EcuSil -  Temperature Low";
  gc_ErrTranslation_fr_Text18 : WSTRING(32) := " [-]: EcuSil -  Temperature High";
  gc_ErrTranslation_fr_Text19 : WSTRING(42) := " [-]: SensorSupply -  Sensor Supply S1 Low";
  gc_ErrTranslation_fr_Text20 : WSTRING(43) := " [-]: SensorSupply -  Sensor Supply S1 High";
  gc_ErrTranslation_fr_Text21 : WSTRING(42) := " [-]: SensorSupply -  Sensor Supply S2 Low";
  gc_ErrTranslation_fr_Text22 : WSTRING(43) := " [-]: SensorSupply -  Sensor Supply S2 High";
  gc_ErrTranslation_fr_Text23 : WSTRING(42) := " [-]: SensorSupply -  Sensor Supply 5V Low";
  gc_ErrTranslation_fr_Text24 : WSTRING(43) := " [-]: SensorSupply -  Sensor Supply 5V High";
  gc_ErrTranslation_fr_Text25 : WSTRING(33) := " [-]: ErrList -  List load oneset";
  gc_ErrTranslation_fr_Text26 : WSTRING(33) := " [-]: ErrList -  List load defect";
  gc_ErrTranslation_fr_Text27 : WSTRING(34) := " [-]: ErrList -  List store defect";
  gc_ErrTranslation_fr_Text28 : WSTRING(29) := " [-]: CAN_BUS0 -  CAN Bus off";
  gc_ErrTranslation_fr_Text29 : WSTRING(29) := " [-]: CAN_BUS0 -  CAN warning";
  gc_ErrTranslation_fr_Text30 : WSTRING(49) := " [-]: CBUS0_HWBUF_SND0 -  HW-Buffer overflow send";
  gc_ErrTranslation_fr_Text31 : WSTRING(49) := " [-]: CBUS0_HWBUF_SND0 -  HW-Buffer overflow send";
  gc_ErrTranslation_fr_Text32 : WSTRING(49) := " [-]: CBUS0_HWBUF_SND0 -  HW-Buffer overflow send";
  gc_ErrTranslation_fr_Text33 : WSTRING(49) := " [-]: CBUS0_HWBUF_SND0 -  HW-Buffer overflow send";
  gc_ErrTranslation_fr_Text34 : WSTRING(49) := " [-]: CBUS0_HWBUF_SND0 -  HW-Buffer overflow send";
  gc_ErrTranslation_fr_Text35 : WSTRING(49) := " [-]: CBUS0_HWBUF_SND0 -  HW-Buffer overflow send";
  gc_ErrTranslation_fr_Text36 : WSTRING(52) := " [-]: CBUS0_HWBUF_RCV0 -  HW-Buffer overflow receive";
  gc_ErrTranslation_fr_Text37 : WSTRING(52) := " [-]: CBUS0_HWBUF_RCV1 -  HW-Buffer overflow receive";
  gc_ErrTranslation_fr_Text38 : WSTRING(52) := " [-]: CBUS0_HWBUF_RCV2 -  HW-Buffer overflow receive";
  gc_ErrTranslation_fr_Text39 : WSTRING(52) := " [-]: CBUS0_HWBUF_RCV3 -  HW-Buffer overflow receive";
  gc_ErrTranslation_fr_Text40 : WSTRING(52) := " [-]: CBUS0_HWBUF_RCV4 -  HW-Buffer overflow receive";
  gc_ErrTranslation_fr_Text41 : WSTRING(52) := " [-]: CBUS0_HWBUF_RCV5 -  HW-Buffer overflow receive";
  gc_ErrTranslation_fr_Text42 : WSTRING(52) := " [-]: CBUS0_HWBUF_RCV6 -  HW-Buffer overflow receive";
  gc_ErrTranslation_fr_Text43 : WSTRING(52) := " [-]: CBUS0_HWBUF_RCV7 -  HW-Buffer overflow receive";
  gc_ErrTranslation_fr_Text44 : WSTRING(40) := " [-]: Ecu0_Safety -  DM_ECU0_INPBOARDNON";
  gc_ErrTranslation_fr_Text45 : WSTRING(40) := " [-]: Ecu0_Safety -  DM_ECU0_INPBOARDFAT";
  gc_ErrTranslation_fr_Text46 : WSTRING(38) := " [-]: Ecu0_Safety -  DM_ECU0_INPUTPINS";
  gc_ErrTranslation_fr_Text47 : WSTRING(67) := " [-]: Ecu0_Safety -  Digital pin error - check ECU hardware and EMI";
  gc_ErrTranslation_fr_Text48 : WSTRING(66) := " [-]: Ecu0_Safety -  PWM output error - check ECU hardware and EMI";
  gc_ErrTranslation_fr_Text49 : WSTRING(63) := " [-]: Ecu0_Safety -  CPU core error - check source code and EMI";
  gc_ErrTranslation_fr_Text50 : WSTRING(33) := " [-]: Ecu0_Safety -  Memory error";
  gc_ErrTranslation_fr_Text51 : WSTRING(86) := " [-]: Ecu0_Safety -  Error during watchdog startup - check watchdog timing constraints";
  gc_ErrTranslation_fr_Text52 : WSTRING(88) := " [-]: Ecu1_Safety -  Safety switch error - check external shut-off pins and ECU hardware";
  gc_ErrTranslation_fr_Text53 : WSTRING(55) := " [-]: Ecu1_Safety -  Application code called safe state";
  gc_ErrTranslation_fr_Text54 : WSTRING(65) := " [-]: Ecu1_Safety -  Fatal error caused safe state -  replace ECU";
  gc_ErrTranslation_fr_Text55 : WSTRING(62) := " [-]: Ecu1_Safety -  BSP error caused safe state - replace ECU";
  gc_ErrTranslation_fr_Text56 : WSTRING(29) := " [-]: EcuSil -  Task overload";
  gc_ErrTranslation_fr_Text57 : WSTRING(28) := " [-]: EcuSil -  Batttery Low";
  gc_ErrTranslation_fr_Text58 : WSTRING(28) := " [-]: EcuSil -  Battery High";
  gc_ErrTranslation_fr_Text59 : WSTRING(31) := " [-]: EcuSil -  Temperature Low";
  gc_ErrTranslation_fr_Text60 : WSTRING(32) := " [-]: EcuSil -  Temperature High";
  gc_ErrTranslation_fr_Text61 : WSTRING(42) := " [-]: SensorSupply -  Sensor Supply S1 Low";
  gc_ErrTranslation_fr_Text62 : WSTRING(43) := " [-]: SensorSupply -  Sensor Supply S1 High";
  gc_ErrTranslation_fr_Text63 : WSTRING(42) := " [-]: SensorSupply -  Sensor Supply S2 Low";
  gc_ErrTranslation_fr_Text64 : WSTRING(43) := " [-]: SensorSupply -  Sensor Supply S2 High";
  gc_ErrTranslation_fr_Text65 : WSTRING(42) := " [-]: SensorSupply -  Sensor Supply 5V Low";
  gc_ErrTranslation_fr_Text66 : WSTRING(43) := " [-]: SensorSupply -  Sensor Supply 5V High";
  gc_ErrTranslation_fr_Text67 : WSTRING(33) := " [-]: ErrList -  List load oneset";
  gc_ErrTranslation_fr_Text68 : WSTRING(33) := " [-]: ErrList -  List load defect";
  gc_ErrTranslation_fr_Text69 : WSTRING(34) := " [-]: ErrList -  List store defect";
  gc_ErrTranslation_fr_Text70 : WSTRING(29) := " [-]: CAN_BUS2 -  CAN Bus off";
  gc_ErrTranslation_fr_Text71 : WSTRING(29) := " [-]: CAN_BUS2 -  CAN warning";
  gc_ErrTranslation_fr_Text72 : WSTRING(49) := " [-]: CBUS2_HWBUF_SND0 -  HW-Buffer overflow send";
  gc_ErrTranslation_fr_Text73 : WSTRING(49) := " [-]: CBUS2_HWBUF_SND0 -  HW-Buffer overflow send";
  gc_ErrTranslation_fr_Text74 : WSTRING(49) := " [-]: CBUS2_HWBUF_SND0 -  HW-Buffer overflow send";
  gc_ErrTranslation_fr_Text75 : WSTRING(49) := " [-]: CBUS2_HWBUF_SND0 -  HW-Buffer overflow send";
  gc_ErrTranslation_fr_Text76 : WSTRING(49) := " [-]: CBUS2_HWBUF_SND0 -  HW-Buffer overflow send";
  gc_ErrTranslation_fr_Text77 : WSTRING(49) := " [-]: CBUS2_HWBUF_SND0 -  HW-Buffer overflow send";
  gc_ErrTranslation_fr_Text78 : WSTRING(52) := " [-]: CBUS2_HWBUF_RCV0 -  HW-Buffer overflow receive";
  gc_ErrTranslation_fr_Text79 : WSTRING(52) := " [-]: CBUS2_HWBUF_RCV1 -  HW-Buffer overflow receive";
  gc_ErrTranslation_fr_Text80 : WSTRING(52) := " [-]: CBUS2_HWBUF_RCV2 -  HW-Buffer overflow receive";
  gc_ErrTranslation_fr_Text81 : WSTRING(52) := " [-]: CBUS2_HWBUF_RCV3 -  HW-Buffer overflow receive";
  gc_ErrTranslation_fr_Text82 : WSTRING(52) := " [-]: CBUS2_HWBUF_RCV4 -  HW-Buffer overflow receive";
  gc_ErrTranslation_fr_Text83 : WSTRING(52) := " [-]: CBUS2_HWBUF_RCV5 -  HW-Buffer overflow receive";
  gc_ErrTranslation_fr_Text84 : WSTRING(52) := " [-]: CBUS2_HWBUF_RCV6 -  HW-Buffer overflow receive";
  gc_ErrTranslation_fr_Text85 : WSTRING(52) := " [-]: CBUS2_HWBUF_RCV7 -  HW-Buffer overflow receive";
  gc_ErrTranslation_fr_Text86 : WSTRING(0) := "";
  gc_ErrTranslation_fr_Text87 : WSTRING(0) := "";
  gc_ErrTranslation_fr_Text88 : WSTRING(0) := "";
  gc_ErrTranslation_fr_Text89 : WSTRING(0) := "";
  gc_ErrTranslation_fr_Text90 : WSTRING(0) := "";
  gc_ErrTranslation_fr_Text91 : WSTRING(0) := "";
  gc_ErrTranslation_fr_Text92 : WSTRING(0) := "";
  gc_ErrTranslation_fr_Text93 : WSTRING(0) := "";
  gc_ErrTranslation_fr_Text94 : WSTRING(0) := "";
  gc_ErrTranslation_fr_Text95 : WSTRING(0) := "";
  gc_ErrTranslation_fr_Text96 : WSTRING(0) := "";
  gc_ErrTranslation_fr_Text97 : WSTRING(0) := "";
  gc_ErrTranslation_fr_Text98 : WSTRING(0) := "";
  gc_ErrTranslation_fr_Text99 : WSTRING(0) := "";
  gc_ErrTranslation_fr_Text100 : WSTRING(0) := "";
  gc_ErrTranslation_fr_Text101 : WSTRING(0) := "";
  gc_ErrTranslation_fr_Text102 : WSTRING(0) := "";
  gc_ErrTranslation_fr_Text103 : WSTRING(0) := "";
  gc_ErrTranslation_fr_Text104 : WSTRING(29) := " [-]: CAN_BUS3 -  CAN Bus off";
  gc_ErrTranslation_fr_Text105 : WSTRING(29) := " [-]: CAN_BUS3 -  CAN warning";
  gc_ErrTranslation_fr_Text106 : WSTRING(49) := " [-]: CBUS3_HWBUF_SND0 -  HW-Buffer overflow send";
  gc_ErrTranslation_fr_Text107 : WSTRING(49) := " [-]: CBUS3_HWBUF_SND0 -  HW-Buffer overflow send";
  gc_ErrTranslation_fr_Text108 : WSTRING(49) := " [-]: CBUS3_HWBUF_SND0 -  HW-Buffer overflow send";
  gc_ErrTranslation_fr_Text109 : WSTRING(49) := " [-]: CBUS3_HWBUF_SND0 -  HW-Buffer overflow send";
  gc_ErrTranslation_fr_Text110 : WSTRING(49) := " [-]: CBUS3_HWBUF_SND0 -  HW-Buffer overflow send";
  gc_ErrTranslation_fr_Text111 : WSTRING(49) := " [-]: CBUS3_HWBUF_SND0 -  HW-Buffer overflow send";
  gc_ErrTranslation_fr_Text112 : WSTRING(52) := " [-]: CBUS3_HWBUF_RCV0 -  HW-Buffer overflow receive";
  gc_ErrTranslation_fr_Text113 : WSTRING(52) := " [-]: CBUS3_HWBUF_RCV1 -  HW-Buffer overflow receive";
  gc_ErrTranslation_fr_Text114 : WSTRING(52) := " [-]: CBUS3_HWBUF_RCV2 -  HW-Buffer overflow receive";
  gc_ErrTranslation_fr_Text115 : WSTRING(52) := " [-]: CBUS3_HWBUF_RCV3 -  HW-Buffer overflow receive";
  gc_ErrTranslation_fr_Text116 : WSTRING(52) := " [-]: CBUS3_HWBUF_RCV4 -  HW-Buffer overflow receive";
  gc_ErrTranslation_fr_Text117 : WSTRING(52) := " [-]: CBUS3_HWBUF_RCV5 -  HW-Buffer overflow receive";
  gc_ErrTranslation_fr_Text118 : WSTRING(52) := " [-]: CBUS3_HWBUF_RCV6 -  HW-Buffer overflow receive";
  gc_ErrTranslation_fr_Text119 : WSTRING(52) := " [-]: CBUS3_HWBUF_RCV7 -  HW-Buffer overflow receive";
  gc_ErrTranslation_fr_Text120 : WSTRING(0) := "";
  gc_ErrTranslation_fr_Text121 : WSTRING(0) := "";
  gc_ErrTranslation_fr_Text122 : WSTRING(6) := " [-]: ";
  gc_ErrTranslation_fr_Text123 : WSTRING(23) := "Message Buffer Overflow";
  gc_ErrTranslation_fr_Text124 : WSTRING(29) := " [-]: CAN_BUS2 -  CAN Bus off";
  gc_ErrTranslation_fr_Text125 : WSTRING(29) := " [-]: CAN_BUS2 -  CAN warning";
  gc_ErrTranslation_fr_Text126 : WSTRING(49) := " [-]: CBUS2_HWBUF_SND0 -  HW-Buffer overflow send";
  gc_ErrTranslation_fr_Text127 : WSTRING(49) := " [-]: CBUS2_HWBUF_SND0 -  HW-Buffer overflow send";
  gc_ErrTranslation_fr_Text128 : WSTRING(49) := " [-]: CBUS2_HWBUF_SND0 -  HW-Buffer overflow send";
  gc_ErrTranslation_fr_Text129 : WSTRING(49) := " [-]: CBUS2_HWBUF_SND0 -  HW-Buffer overflow send";
  gc_ErrTranslation_fr_Text130 : WSTRING(49) := " [-]: CBUS2_HWBUF_SND0 -  HW-Buffer overflow send";
  gc_ErrTranslation_fr_Text131 : WSTRING(49) := " [-]: CBUS2_HWBUF_SND0 -  HW-Buffer overflow send";
  gc_ErrTranslation_fr_Text132 : WSTRING(52) := " [-]: CBUS2_HWBUF_RCV0 -  HW-Buffer overflow receive";
  gc_ErrTranslation_fr_Text133 : WSTRING(52) := " [-]: CBUS2_HWBUF_RCV1 -  HW-Buffer overflow receive";
  gc_ErrTranslation_fr_Text134 : WSTRING(52) := " [-]: CBUS2_HWBUF_RCV2 -  HW-Buffer overflow receive";
  gc_ErrTranslation_fr_Text135 : WSTRING(52) := " [-]: CBUS2_HWBUF_RCV3 -  HW-Buffer overflow receive";
  gc_ErrTranslation_fr_Text136 : WSTRING(52) := " [-]: CBUS2_HWBUF_RCV4 -  HW-Buffer overflow receive";
  gc_ErrTranslation_fr_Text137 : WSTRING(52) := " [-]: CBUS2_HWBUF_RCV5 -  HW-Buffer overflow receive";
  gc_ErrTranslation_fr_Text138 : WSTRING(52) := " [-]: CBUS2_HWBUF_RCV6 -  HW-Buffer overflow receive";
  gc_ErrTranslation_fr_Text139 : WSTRING(52) := " [-]: CBUS2_HWBUF_RCV7 -  HW-Buffer overflow receive";
  gc_ErrTranslation_fr_Text140 : WSTRING(0) := "";
  gc_ErrTranslation_fr_Text141 : WSTRING(0) := "";
  gc_ErrTranslation_fr_Text142 : WSTRING(49) := " [-]: CBUS0_HWBUF_SND0 -  HW-Buffer overflow send";
  gc_ErrTranslation_fr_Text143 : WSTRING(49) := " [-]: CBUS0_HWBUF_SND0 -  HW-Buffer overflow send";
  gc_ErrTranslation_fr_Text144 : WSTRING(49) := " [-]: CBUS0_HWBUF_SND0 -  HW-Buffer overflow send";
  gc_ErrTranslation_fr_Text145 : WSTRING(49) := " [-]: CBUS0_HWBUF_SND0 -  HW-Buffer overflow send";
  gc_ErrTranslation_fr_Text146 : WSTRING(49) := " [-]: CBUS0_HWBUF_SND0 -  HW-Buffer overflow send";
  gc_ErrTranslation_fr_Text147 : WSTRING(49) := " [-]: CBUS0_HWBUF_SND0 -  HW-Buffer overflow send";
  gc_ErrTranslation_fr_Text148 : WSTRING(52) := " [-]: CBUS0_HWBUF_RCV0 -  HW-Buffer overflow receive";
  gc_ErrTranslation_fr_Text149 : WSTRING(52) := " [-]: CBUS0_HWBUF_RCV1 -  HW-Buffer overflow receive";
  gc_ErrTranslation_fr_Text150 : WSTRING(52) := " [-]: CBUS0_HWBUF_RCV2 -  HW-Buffer overflow receive";
  gc_ErrTranslation_fr_Text151 : WSTRING(52) := " [-]: CBUS0_HWBUF_RCV3 -  HW-Buffer overflow receive";
  gc_ErrTranslation_fr_Text152 : WSTRING(52) := " [-]: CBUS0_HWBUF_RCV4 -  HW-Buffer overflow receive";
  gc_ErrTranslation_fr_Text153 : WSTRING(52) := " [-]: CBUS0_HWBUF_RCV5 -  HW-Buffer overflow receive";
  gc_ErrTranslation_fr_Text154 : WSTRING(52) := " [-]: CBUS0_HWBUF_RCV6 -  HW-Buffer overflow receive";
  gc_ErrTranslation_fr_Text155 : WSTRING(52) := " [-]: CBUS0_HWBUF_RCV7 -  HW-Buffer overflow receive";
  gc_ErrTranslation_fr_Text156 : WSTRING(26) := "Time out of cyclic message";
  gc_ErrTranslation_fr_Text157 : WSTRING(23) := "Message Buffer Overflow";
  gc_ErrTranslation_fr_Text158 : WSTRING(15) := "Invalid Message";
  gc_ErrTranslation_fr_Text159 : WSTRING(11) := "Count Fault";
  gc_ErrTranslation_fr_Text160 : WSTRING(8) := "Timeslot";
  gc_ErrTranslation_fr_Text161 : WSTRING(26) := "Time out of cyclic message";
  gc_ErrTranslation_fr_Text162 : WSTRING(23) := "Message Buffer Overflow";
  gc_ErrTranslation_fr_Text163 : WSTRING(15) := "Invalid Message";
  gc_ErrTranslation_fr_Text164 : WSTRING(11) := "Count Fault";
  gc_ErrTranslation_fr_Text165 : WSTRING(8) := "Timeslot";
  gc_ErrTranslation_fr_Text166 : WSTRING(26) := "Time out of cyclic message";
  gc_ErrTranslation_fr_Text167 : WSTRING(23) := "Message Buffer Overflow";
  gc_ErrTranslation_fr_Text168 : WSTRING(15) := "Invalid Message";
  gc_ErrTranslation_fr_Text169 : WSTRING(11) := "Count Fault";
  gc_ErrTranslation_fr_Text170 : WSTRING(8) := "Timeslot";
  gc_ErrTranslation_fr_Text171 : WSTRING(26) := "Time out of cyclic message";
  gc_ErrTranslation_fr_Text172 : WSTRING(23) := "Message Buffer Overflow";
  gc_ErrTranslation_fr_Text173 : WSTRING(15) := "Invalid Message";
  gc_ErrTranslation_fr_Text174 : WSTRING(11) := "Count Fault";
  gc_ErrTranslation_fr_Text175 : WSTRING(8) := "Timeslot";
  gc_ErrTranslation_fr_Text176 : WSTRING(26) := "Time out of cyclic message";
  gc_ErrTranslation_fr_Text177 : WSTRING(23) := "Message Buffer Overflow";
  gc_ErrTranslation_fr_Text178 : WSTRING(15) := "Invalid Message";
  gc_ErrTranslation_fr_Text179 : WSTRING(11) := "Count Fault";
  gc_ErrTranslation_fr_Text180 : WSTRING(29) := " [-]: CAN_BUS1 -  CAN Bus off";
  gc_ErrTranslation_fr_Text181 : WSTRING(29) := " [-]: CAN_BUS1 -  CAN warning";
  gc_ErrTranslation_fr_Text182 : WSTRING(49) := " [-]: CBUS1_HWBUF_SND0 -  HW-Buffer overflow send";
  gc_ErrTranslation_fr_Text183 : WSTRING(49) := " [-]: CBUS1_HWBUF_SND0 -  HW-Buffer overflow send";
  gc_ErrTranslation_fr_Text184 : WSTRING(49) := " [-]: CBUS1_HWBUF_SND0 -  HW-Buffer overflow send";
  gc_ErrTranslation_fr_Text185 : WSTRING(49) := " [-]: CBUS1_HWBUF_SND0 -  HW-Buffer overflow send";
  gc_ErrTranslation_fr_Text186 : WSTRING(49) := " [-]: CBUS1_HWBUF_SND0 -  HW-Buffer overflow send";
  gc_ErrTranslation_fr_Text187 : WSTRING(49) := " [-]: CBUS1_HWBUF_SND0 -  HW-Buffer overflow send";
  gc_ErrTranslation_fr_Text188 : WSTRING(52) := " [-]: CBUS1_HWBUF_RCV0 -  HW-Buffer overflow receive";
  gc_ErrTranslation_fr_Text189 : WSTRING(52) := " [-]: CBUS1_HWBUF_RCV1 -  HW-Buffer overflow receive";
  gc_ErrTranslation_fr_Text190 : WSTRING(52) := " [-]: CBUS1_HWBUF_RCV2 -  HW-Buffer overflow receive";
  gc_ErrTranslation_fr_Text191 : WSTRING(52) := " [-]: CBUS1_HWBUF_RCV3 -  HW-Buffer overflow receive";
  gc_ErrTranslation_fr_Text192 : WSTRING(52) := " [-]: CBUS1_HWBUF_RCV4 -  HW-Buffer overflow receive";
  gc_ErrTranslation_fr_Text193 : WSTRING(52) := " [-]: CBUS1_HWBUF_RCV5 -  HW-Buffer overflow receive";
  gc_ErrTranslation_fr_Text194 : WSTRING(52) := " [-]: CBUS1_HWBUF_RCV6 -  HW-Buffer overflow receive";
  gc_ErrTranslation_fr_Text195 : WSTRING(52) := " [-]: CBUS1_HWBUF_RCV7 -  HW-Buffer overflow receive";
  gc_ErrTranslation_fr_Text196 : WSTRING(29) := " [-]: CAN_BUS1 -  CAN Bus off";
  gc_ErrTranslation_fr_Text197 : WSTRING(29) := " [-]: CAN_BUS1 -  CAN warning";
  gc_ErrTranslation_fr_Text198 : WSTRING(49) := " [-]: CBUS1_HWBUF_SND0 -  HW-Buffer overflow send";
  gc_ErrTranslation_fr_Text199 : WSTRING(49) := " [-]: CBUS1_HWBUF_SND0 -  HW-Buffer overflow send";
  gc_ErrTranslation_fr_Text200 : WSTRING(49) := " [-]: CBUS1_HWBUF_SND0 -  HW-Buffer overflow send";
  gc_ErrTranslation_fr_Text201 : WSTRING(49) := " [-]: CBUS1_HWBUF_SND0 -  HW-Buffer overflow send";
  gc_ErrTranslation_fr_Text202 : WSTRING(49) := " [-]: CBUS1_HWBUF_SND0 -  HW-Buffer overflow send";
  gc_ErrTranslation_fr_Text203 : WSTRING(49) := " [-]: CBUS1_HWBUF_SND0 -  HW-Buffer overflow send";
  gc_ErrTranslation_fr_Text204 : WSTRING(52) := " [-]: CBUS1_HWBUF_RCV0 -  HW-Buffer overflow receive";
  gc_ErrTranslation_fr_Text205 : WSTRING(52) := " [-]: CBUS1_HWBUF_RCV1 -  HW-Buffer overflow receive";
  gc_ErrTranslation_fr_Text206 : WSTRING(52) := " [-]: CBUS1_HWBUF_RCV2 -  HW-Buffer overflow receive";
  gc_ErrTranslation_fr_Text207 : WSTRING(52) := " [-]: CBUS1_HWBUF_RCV3 -  HW-Buffer overflow receive";
  gc_ErrTranslation_fr_Text208 : WSTRING(52) := " [-]: CBUS1_HWBUF_RCV4 -  HW-Buffer overflow receive";
  gc_ErrTranslation_fr_Text209 : WSTRING(52) := " [-]: CBUS1_HWBUF_RCV5 -  HW-Buffer overflow receive";
  gc_ErrTranslation_fr_Text210 : WSTRING(52) := " [-]: CBUS1_HWBUF_RCV6 -  HW-Buffer overflow receive";
  gc_ErrTranslation_fr_Text211 : WSTRING(52) := " [-]: CBUS1_HWBUF_RCV7 -  HW-Buffer overflow receive";
  gc_ErrTranslation_fr_Text212 : WSTRING(8) := "Timeslot";
  gc_ErrTranslation_fr_Text213 : WSTRING(26) := "Time out of cyclic message";
  gc_ErrTranslation_fr_Text214 : WSTRING(23) := "Message Buffer Overflow";
  gc_ErrTranslation_fr_Text215 : WSTRING(15) := "Invalid Message";
  gc_ErrTranslation_fr_Text216 : WSTRING(11) := "Count Fault";
  gc_ErrTranslation_fr_Text217 : WSTRING(8) := "Timeslot";
  gc_ErrTranslation_fr_Text218 : WSTRING(18) := "DMx protocol error";
  gc_ErrTranslation_fr_Text219 : WSTRING(16) := "CAN Snd Overflow";
  gc_ErrTranslation_fr_Text220 : WSTRING(18) := "DMx protocol error";
  gc_ErrTranslation_fr_Text221 : WSTRING(16) := "CAN Snd Overflow";
  gc_ErrTranslation_fr_Text222 : WSTRING(0) := "";
  gc_ErrTranslation_fr_Text223 : WSTRING(0) := "";
  gc_ErrTranslation_fr_Text224 : WSTRING(0) := "";
  gc_ErrTranslation_fr_Text225 : WSTRING(23) := "Message buffer overflow";
  gc_ErrTranslation_fr_Text226 : WSTRING(26) := "Time out of cyclic message";
  gc_ErrTranslation_fr_Text227 : WSTRING(23) := "Message buffer overflow";
  gc_ErrTranslation_fr_Text228 : WSTRING(15) := "Invalid message";
  gc_ErrTranslation_fr_Text229 : WSTRING(11) := "Count fault";
  gc_ErrTranslation_fr_Text230 : WSTRING(8) := "Timeslot";
  gc_ErrTranslation_fr_Text231 : WSTRING(26) := "Time out of cyclic message";
  gc_ErrTranslation_fr_Text232 : WSTRING(23) := "Message buffer overflow";
  gc_ErrTranslation_fr_Text233 : WSTRING(15) := "Invalid message";
  gc_ErrTranslation_fr_Text234 : WSTRING(11) := "Count fault";
  gc_ErrTranslation_fr_Text235 : WSTRING(8) := "Timeslot";
  gc_ErrTranslation_fr_Text236 : WSTRING(23) := "Message buffer overflow";
  gc_ErrTranslation_fr_Text237 : WSTRING(0) := "";
  gc_ErrTranslation_fr_Text238 : WSTRING(0) := "";
  gc_ErrTranslation_fr_Text239 : WSTRING(0) := "";
  gc_ErrTranslation_fr_Text240 : WSTRING(26) := "Time out of cyclic message";
  gc_ErrTranslation_fr_Text241 : WSTRING(23) := "Message buffer overflow";
  gc_ErrTranslation_fr_Text242 : WSTRING(15) := "Invalid message";
  gc_ErrTranslation_fr_Text243 : WSTRING(11) := "Count fault";
  gc_ErrTranslation_fr_Text244 : WSTRING(8) := "Timeslot";
  gc_ErrTranslation_fr_Text245 : WSTRING(26) := "Time out of cyclic message";
  gc_ErrTranslation_fr_Text246 : WSTRING(23) := "Message buffer overflow";
  gc_ErrTranslation_fr_Text247 : WSTRING(15) := "Invalid message";
  gc_ErrTranslation_fr_Text248 : WSTRING(11) := "Count fault";
  gc_ErrTranslation_fr_Text249 : WSTRING(8) := "Timeslot";
  gc_ErrTranslation_fr_Text250 : WSTRING(26) := "Time out of cyclic message";
  gc_ErrTranslation_fr_Text251 : WSTRING(23) := "Message buffer overflow";
  gc_ErrTranslation_fr_Text252 : WSTRING(15) := "Invalid message";
  gc_ErrTranslation_fr_Text253 : WSTRING(11) := "Count fault";
  gc_ErrTranslation_fr_Text254 : WSTRING(8) := "Timeslot";
  gc_ErrTranslation_fr_Text255 : WSTRING(26) := "Time out of cyclic message";
  gc_ErrTranslation_fr_Text256 : WSTRING(23) := "Message buffer overflow";
  gc_ErrTranslation_fr_Text257 : WSTRING(15) := "Invalid message";
  gc_ErrTranslation_fr_Text258 : WSTRING(11) := "Count fault";
  gc_ErrTranslation_fr_Text259 : WSTRING(8) := "Timeslot";
  gc_ErrTranslation_fr_Text260 : WSTRING(26) := "Time out of cyclic message";
  gc_ErrTranslation_fr_Text261 : WSTRING(23) := "Message buffer overflow";
  gc_ErrTranslation_fr_Text262 : WSTRING(15) := "Invalid message";
  gc_ErrTranslation_fr_Text263 : WSTRING(11) := "Count fault";
  gc_ErrTranslation_fr_Text264 : WSTRING(8) := "Timeslot";
  gc_ErrTranslation_fr_Text265 : WSTRING(23) := "Message buffer overflow";
  gc_ErrTranslation_fr_Text266 : WSTRING(23) := "Message buffer overflow";
  gc_ErrTranslation_fr_Text267 : WSTRING(23) := "Message buffer overflow";
  gc_ErrTranslation_fr_Text268 : WSTRING(23) := "Message buffer overflow";
  gc_ErrTranslation_fr_Text269 : WSTRING(23) := "Message buffer overflow";
  gc_ErrTranslation_fr_Text270 : WSTRING(23) := "Message buffer overflow";
  gc_ErrTranslation_fr_Text271 : WSTRING(23) := "Message buffer overflow";
  gc_ErrTranslation_fr_Text272 : WSTRING(23) := "Message buffer overflow";
  gc_ErrTranslation_fr_Text273 : WSTRING(26) := "Time out of cyclic message";
  gc_ErrTranslation_fr_Text274 : WSTRING(23) := "Message buffer overflow";
  gc_ErrTranslation_fr_Text275 : WSTRING(15) := "Invalid message";
  gc_ErrTranslation_fr_Text276 : WSTRING(11) := "Count fault";
  gc_ErrTranslation_fr_Text277 : WSTRING(8) := "Timeslot";
  gc_ErrTranslation_fr_Text278 : WSTRING(23) := "Message buffer overflow";
  gc_ErrTranslation_fr_Text279 : WSTRING(26) := "Time out of cyclic message";
  gc_ErrTranslation_fr_Text280 : WSTRING(23) := "Message buffer overflow";
  gc_ErrTranslation_fr_Text281 : WSTRING(15) := "Invalid message";
  gc_ErrTranslation_fr_Text282 : WSTRING(11) := "Count fault";
  gc_ErrTranslation_fr_Text283 : WSTRING(8) := "Timeslot";
  gc_ErrTranslation_fr_Text284 : WSTRING(23) := "Message buffer overflow";
  gc_ErrTranslation_fr_Text285 : WSTRING(26) := "Time out of cyclic message";
  gc_ErrTranslation_fr_Text286 : WSTRING(23) := "Message buffer overflow";
  gc_ErrTranslation_fr_Text287 : WSTRING(15) := "Invalid message";
  gc_ErrTranslation_fr_Text288 : WSTRING(11) := "Count fault";
  gc_ErrTranslation_fr_Text289 : WSTRING(8) := "Timeslot";
  gc_ErrTranslation_fr_Text290 : WSTRING(26) := "Time out of cyclic message";
  gc_ErrTranslation_fr_Text291 : WSTRING(23) := "Message buffer overflow";
  gc_ErrTranslation_fr_Text292 : WSTRING(15) := "Invalid message";
  gc_ErrTranslation_fr_Text293 : WSTRING(11) := "Count fault";
  gc_ErrTranslation_fr_Text294 : WSTRING(8) := "Timeslot";
  gc_ErrTranslation_fr_Text295 : WSTRING(26) := "Time out of cyclic message";
  gc_ErrTranslation_fr_Text296 : WSTRING(23) := "Message buffer overflow";
  gc_ErrTranslation_fr_Text297 : WSTRING(15) := "Invalid message";
  gc_ErrTranslation_fr_Text298 : WSTRING(11) := "Count fault";
  gc_ErrTranslation_fr_Text299 : WSTRING(8) := "Timeslot";
  gc_ErrTranslation_fr_Text300 : WSTRING(23) := "Message buffer overflow";
  gc_ErrTranslation_fr_Text301 : WSTRING(23) := "Message buffer overflow";
  gc_ErrTranslation_fr_Text302 : WSTRING(81) := " [PIN_103 ]: PressureBlockOscillationSensor -  Master input signal short to power";
  gc_ErrTranslation_fr_Text303 : WSTRING(82) := " [PIN_103 ]: PressureBlockOscillationSensor -  Master input signal short to ground";
  gc_ErrTranslation_fr_Text304 : WSTRING(82) := " [PIN_103 ]: PressureBlockOscillationSensor -  Parameter of input char NOT monoton";
  gc_ErrTranslation_fr_Text305 : WSTRING(69) := " [PIN_103 ]: PressureBlockOscillationSensor -  Unknown internal error";
  gc_ErrTranslation_fr_Text306 : WSTRING(70) := " [PIN_127 ]: PressureBrakeSensor -  Master input signal short to power";
  gc_ErrTranslation_fr_Text307 : WSTRING(71) := " [PIN_127 ]: PressureBrakeSensor -  Master input signal short to ground";
  gc_ErrTranslation_fr_Text308 : WSTRING(71) := " [PIN_127 ]: PressureBrakeSensor -  Parameter of input char NOT monoton";
  gc_ErrTranslation_fr_Text309 : WSTRING(58) := " [PIN_127 ]: PressureBrakeSensor -  Unknown internal error";
  gc_ErrTranslation_fr_Text310 : WSTRING(78) := " [PIN_103 ]: Transmission1PressureSensor -  Master input signal short to power";
  gc_ErrTranslation_fr_Text311 : WSTRING(79) := " [PIN_103 ]: Transmission1PressureSensor -  Master input signal short to ground";
  gc_ErrTranslation_fr_Text312 : WSTRING(79) := " [PIN_103 ]: Transmission1PressureSensor -  Parameter of input char NOT monoton";
  gc_ErrTranslation_fr_Text313 : WSTRING(66) := " [PIN_103 ]: Transmission1PressureSensor -  Unknown internal error";
  gc_ErrTranslation_fr_Text314 : WSTRING(27) := " [-]: SpecificErrorC0_5 -  ";
  gc_ErrTranslation_fr_Text315 : WSTRING(27) := " [-]: SpecificErrorC0_5 -  ";
  gc_ErrTranslation_fr_Text316 : WSTRING(77) := " [-]: SpecificErrorC0_5 -  Check pressure when bypass is pilot detected by C1";
  gc_ErrTranslation_fr_Text317 : WSTRING(27) := " [-]: SpecificErrorC0_5 -  ";
  gc_ErrTranslation_fr_Text318 : WSTRING(38) := " [-]: SpecificErrorC0_5 -  Error bit 4";
  gc_ErrTranslation_fr_Text319 : WSTRING(38) := " [-]: SpecificErrorC0_5 -  Error bit 5";
  gc_ErrTranslation_fr_Text320 : WSTRING(38) := " [-]: SpecificErrorC0_5 -  Error bit 6";
  gc_ErrTranslation_fr_Text321 : WSTRING(10) := "DMC erreur";
  gc_ErrTranslation_fr_Text322 : WSTRING(65) := " [PIN_115 ]: OscillantAxleSpeedSensor -  Input is short to Ground";
  gc_ErrTranslation_fr_Text323 : WSTRING(64) := " [PIN_115 ]: OscillantAxleSpeedSensor -  Input is short to Power";
  gc_ErrTranslation_fr_Text324 : WSTRING(56) := " [PIN_115 ]: OscillantAxleSpeedSensor -  Wrong Parameter";
  gc_ErrTranslation_fr_Text325 : WSTRING(54) := " [PIN_115 ]: OscillantAxleSpeedSensor -  Unknown Error";
  gc_ErrTranslation_fr_Text326 : WSTRING(60) := " [PIN_116 ]: FixeAxleSpeedSensor -  Input is short to Ground";
  gc_ErrTranslation_fr_Text327 : WSTRING(59) := " [PIN_116 ]: FixeAxleSpeedSensor -  Input is short to Power";
  gc_ErrTranslation_fr_Text328 : WSTRING(51) := " [PIN_116 ]: FixeAxleSpeedSensor -  Wrong Parameter";
  gc_ErrTranslation_fr_Text329 : WSTRING(49) := " [PIN_116 ]: FixeAxleSpeedSensor -  Unknown Error";
  gc_ErrTranslation_fr_Text330 : WSTRING(77) := " [PIN_153 ]: EvDeflectorTransmission -  HS OpenLoad / Short To Power external";
  gc_ErrTranslation_fr_Text331 : WSTRING(66) := " [PIN_153 ]: EvDeflectorTransmission -  HS Short To Power internal";
  gc_ErrTranslation_fr_Text332 : WSTRING(58) := " [PIN_153 ]: EvDeflectorTransmission -  HS Short To Ground";
  gc_ErrTranslation_fr_Text333 : WSTRING(61) := " [PIN_153 ]: EvDeflectorTransmission -  Internal Driver Error";
  gc_ErrTranslation_fr_Text334 : WSTRING(71) := " [PIN_190 ]: EvUpMeasuringMast -  HS OpenLoad / Short To Power external";
  gc_ErrTranslation_fr_Text335 : WSTRING(60) := " [PIN_190 ]: EvUpMeasuringMast -  HS Short To Power internal";
  gc_ErrTranslation_fr_Text336 : WSTRING(52) := " [PIN_190 ]: EvUpMeasuringMast -  HS Short To Ground";
  gc_ErrTranslation_fr_Text337 : WSTRING(55) := " [PIN_190 ]: EvUpMeasuringMast -  Internal Driver Error";
  gc_ErrTranslation_fr_Text338 : WSTRING(73) := " [PIN_166 ]: EvDownMeasuringMast -  HS OpenLoad / Short To Power external";
  gc_ErrTranslation_fr_Text339 : WSTRING(62) := " [PIN_166 ]: EvDownMeasuringMast -  HS Short To Power internal";
  gc_ErrTranslation_fr_Text340 : WSTRING(54) := " [PIN_166 ]: EvDownMeasuringMast -  HS Short To Ground";
  gc_ErrTranslation_fr_Text341 : WSTRING(57) := " [PIN_166 ]: EvDownMeasuringMast -  Internal Driver Error";
  gc_ErrTranslation_fr_Text342 : WSTRING(73) := " [PIN_195 ]: EvServiceBrakeTrack -  HS OpenLoad / Short To Power external";
  gc_ErrTranslation_fr_Text343 : WSTRING(62) := " [PIN_195 ]: EvServiceBrakeTrack -  HS Short To Power internal";
  gc_ErrTranslation_fr_Text344 : WSTRING(54) := " [PIN_195 ]: EvServiceBrakeTrack -  HS Short To Ground";
  gc_ErrTranslation_fr_Text345 : WSTRING(57) := " [PIN_195 ]: EvServiceBrakeTrack -  Internal Driver Error";
  gc_ErrTranslation_fr_Text346 : WSTRING(70) := " [PIN_171 ]: EvPowerReduction -  HS OpenLoad / Short To Power external";
  gc_ErrTranslation_fr_Text347 : WSTRING(59) := " [PIN_171 ]: EvPowerReduction -  HS Short To Power internal";
  gc_ErrTranslation_fr_Text348 : WSTRING(51) := " [PIN_171 ]: EvPowerReduction -  HS Short To Ground";
  gc_ErrTranslation_fr_Text349 : WSTRING(54) := " [PIN_171 ]: EvPowerReduction -  Internal Driver Error";
  gc_ErrTranslation_fr_Text350 : WSTRING(78) := " [PIN_127 ]: Transmission2PressureSensor -  Master input signal short to power";
  gc_ErrTranslation_fr_Text351 : WSTRING(79) := " [PIN_127 ]: Transmission2PressureSensor -  Master input signal short to ground";
  gc_ErrTranslation_fr_Text352 : WSTRING(79) := " [PIN_127 ]: Transmission2PressureSensor -  Parameter of input char NOT monoton";
  gc_ErrTranslation_fr_Text353 : WSTRING(66) := " [PIN_127 ]: Transmission2PressureSensor -  Unknown internal error";
  gc_ErrTranslation_fr_Text354 : WSTRING(75) := " [PIN_131 PIN_122 ]: DownOscillantAxle -  Logical Error between pin 0 and 1";
  gc_ErrTranslation_fr_Text355 : WSTRING(60) := " [PIN_131 PIN_122 ]: DownOscillantAxle -  Vin0 < u16VolLoMin";
  gc_ErrTranslation_fr_Text356 : WSTRING(60) := " [PIN_131 PIN_122 ]: DownOscillantAxle -  Vin0 > u16VolHiMax";
  gc_ErrTranslation_fr_Text357 : WSTRING(74) := " [PIN_131 PIN_122 ]: DownOscillantAxle -  u16VolLoMax < Vin0 < u16VolHiMin";
  gc_ErrTranslation_fr_Text358 : WSTRING(73) := " [PIN_160 ]: SupplyRadioReceiver -  HS OpenLoad / Short To Power external";
  gc_ErrTranslation_fr_Text359 : WSTRING(62) := " [PIN_160 ]: SupplyRadioReceiver -  HS Short To Power internal";
  gc_ErrTranslation_fr_Text360 : WSTRING(54) := " [PIN_160 ]: SupplyRadioReceiver -  HS Short To Ground";
  gc_ErrTranslation_fr_Text361 : WSTRING(57) := " [PIN_160 ]: SupplyRadioReceiver -  Internal Driver Error";
  gc_ErrTranslation_fr_Text362 : WSTRING(77) := " [PIN_184 ]: BuzzerLynxMovingMachine -  HS OpenLoad / Short To Power external";
  gc_ErrTranslation_fr_Text363 : WSTRING(66) := " [PIN_184 ]: BuzzerLynxMovingMachine -  HS Short To Power internal";
  gc_ErrTranslation_fr_Text364 : WSTRING(58) := " [PIN_184 ]: BuzzerLynxMovingMachine -  HS Short To Ground";
  gc_ErrTranslation_fr_Text365 : WSTRING(61) := " [PIN_184 ]: BuzzerLynxMovingMachine -  Internal Driver Error";
  gc_ErrTranslation_fr_Text366 : WSTRING(80) := " [PIN_104 ]: TemperatureTransmissionSensor -  Master input signal short to power";
  gc_ErrTranslation_fr_Text367 : WSTRING(81) := " [PIN_104 ]: TemperatureTransmissionSensor -  Master input signal short to ground";
  gc_ErrTranslation_fr_Text368 : WSTRING(81) := " [PIN_104 ]: TemperatureTransmissionSensor -  Parameter of input char NOT monoton";
  gc_ErrTranslation_fr_Text369 : WSTRING(68) := " [PIN_104 ]: TemperatureTransmissionSensor -  Unknown internal error";
  gc_ErrTranslation_fr_Text370 : WSTRING(66) := " [PIN_150 ]: CoolingRelay -  HS OpenLoad / Short To Power external";
  gc_ErrTranslation_fr_Text371 : WSTRING(55) := " [PIN_150 ]: CoolingRelay -  HS Short To Power internal";
  gc_ErrTranslation_fr_Text372 : WSTRING(47) := " [PIN_150 ]: CoolingRelay -  HS Short To Ground";
  gc_ErrTranslation_fr_Text373 : WSTRING(50) := " [PIN_150 ]: CoolingRelay -  Internal Driver Error";
  gc_ErrTranslation_fr_Text374 : WSTRING(67) := " [PIN_173 ]: WhiteLightAVD -  HS OpenLoad / Short To Power external";
  gc_ErrTranslation_fr_Text375 : WSTRING(56) := " [PIN_173 ]: WhiteLightAVD -  HS Short To Power internal";
  gc_ErrTranslation_fr_Text376 : WSTRING(48) := " [PIN_173 ]: WhiteLightAVD -  HS Short To Ground";
  gc_ErrTranslation_fr_Text377 : WSTRING(51) := " [PIN_173 ]: WhiteLightAVD -  Internal Driver Error";
  gc_ErrTranslation_fr_Text378 : WSTRING(65) := " [PIN_152 ]: RedLightAVG -  HS OpenLoad / Short To Power external";
  gc_ErrTranslation_fr_Text379 : WSTRING(54) := " [PIN_152 ]: RedLightAVG -  HS Short To Power internal";
  gc_ErrTranslation_fr_Text380 : WSTRING(46) := " [PIN_152 ]: RedLightAVG -  HS Short To Ground";
  gc_ErrTranslation_fr_Text381 : WSTRING(49) := " [PIN_152 ]: RedLightAVG -  Internal Driver Error";
  gc_ErrTranslation_fr_Text382 : WSTRING(65) := " [PIN_176 ]: RedLightAVD -  HS OpenLoad / Short To Power external";
  gc_ErrTranslation_fr_Text383 : WSTRING(54) := " [PIN_176 ]: RedLightAVD -  HS Short To Power internal";
  gc_ErrTranslation_fr_Text384 : WSTRING(46) := " [PIN_176 ]: RedLightAVD -  HS Short To Ground";
  gc_ErrTranslation_fr_Text385 : WSTRING(49) := " [PIN_176 ]: RedLightAVD -  Internal Driver Error";
  gc_ErrTranslation_fr_Text386 : WSTRING(67) := " [PIN_155 ]: WhiteLightARG -  HS OpenLoad / Short To Power external";
  gc_ErrTranslation_fr_Text387 : WSTRING(56) := " [PIN_155 ]: WhiteLightARG -  HS Short To Power internal";
  gc_ErrTranslation_fr_Text388 : WSTRING(48) := " [PIN_155 ]: WhiteLightARG -  HS Short To Ground";
  gc_ErrTranslation_fr_Text389 : WSTRING(51) := " [PIN_155 ]: WhiteLightARG -  Internal Driver Error";
  gc_ErrTranslation_fr_Text390 : WSTRING(67) := " [PIN_179 ]: WhiteLightARD -  HS OpenLoad / Short To Power external";
  gc_ErrTranslation_fr_Text391 : WSTRING(56) := " [PIN_179 ]: WhiteLightARD -  HS Short To Power internal";
  gc_ErrTranslation_fr_Text392 : WSTRING(48) := " [PIN_179 ]: WhiteLightARD -  HS Short To Ground";
  gc_ErrTranslation_fr_Text393 : WSTRING(51) := " [PIN_179 ]: WhiteLightARD -  Internal Driver Error";
  gc_ErrTranslation_fr_Text394 : WSTRING(65) := " [PIN_158 ]: RedLightARG -  HS OpenLoad / Short To Power external";
  gc_ErrTranslation_fr_Text395 : WSTRING(54) := " [PIN_158 ]: RedLightARG -  HS Short To Power internal";
  gc_ErrTranslation_fr_Text396 : WSTRING(46) := " [PIN_158 ]: RedLightARG -  HS Short To Ground";
  gc_ErrTranslation_fr_Text397 : WSTRING(49) := " [PIN_158 ]: RedLightARG -  Internal Driver Error";
  gc_ErrTranslation_fr_Text398 : WSTRING(65) := " [PIN_182 ]: RedLightARD -  HS OpenLoad / Short To Power external";
  gc_ErrTranslation_fr_Text399 : WSTRING(54) := " [PIN_182 ]: RedLightARD -  HS Short To Power internal";
  gc_ErrTranslation_fr_Text400 : WSTRING(46) := " [PIN_182 ]: RedLightARD -  HS Short To Ground";
  gc_ErrTranslation_fr_Text401 : WSTRING(49) := " [PIN_182 ]: RedLightARD -  Internal Driver Error";
  gc_ErrTranslation_fr_Text402 : WSTRING(73) := " [PIN_164 ]: SupplyPvgRightTrack -  HS OpenLoad / Short To Power external";
  gc_ErrTranslation_fr_Text403 : WSTRING(62) := " [PIN_164 ]: SupplyPvgRightTrack -  HS Short To Power internal";
  gc_ErrTranslation_fr_Text404 : WSTRING(54) := " [PIN_164 ]: SupplyPvgRightTrack -  HS Short To Ground";
  gc_ErrTranslation_fr_Text405 : WSTRING(57) := " [PIN_164 ]: SupplyPvgRightTrack -  Internal Driver Error";
  gc_ErrTranslation_fr_Text406 : WSTRING(60) := " [PIN_131 PIN_122 ]: DownOscillantAxle -  Vin1 < u16VolLoMin";
  gc_ErrTranslation_fr_Text407 : WSTRING(60) := " [PIN_131 PIN_122 ]: DownOscillantAxle -  Vin1 > u16VolHiMax";
  gc_ErrTranslation_fr_Text408 : WSTRING(74) := " [PIN_131 PIN_122 ]: DownOscillantAxle -  u16VolLoMax < Vin1 < u16VolHiMin";
  gc_ErrTranslation_fr_Text409 : WSTRING(56) := " [-]: SpecificErrorC1_2 -  Coherence pilotage PVG Ev Tor";
  gc_ErrTranslation_fr_Text410 : WSTRING(59) := " [-]: SpecificErrorC1_2 -  Coherence pilotage PVG telescope";
  gc_ErrTranslation_fr_Text411 : WSTRING(52) := "An input signal is too low / Short circuit to ground";
  gc_ErrTranslation_fr_Text412 : WSTRING(52) := "An input signal is too high / Short circuit to power";
  gc_ErrTranslation_fr_Text413 : WSTRING(37) := "An input signal is out of valid range";
  gc_ErrTranslation_fr_Text414 : WSTRING(39) := "Warning: a block has limited parameters";
  gc_ErrTranslation_fr_Text415 : WSTRING(23) := "An initialization error";
  gc_ErrTranslation_fr_Text416 : WSTRING(52) := "An input signal is too low / Short circuit to ground";
  gc_ErrTranslation_fr_Text417 : WSTRING(84) := " [PIN_132 ]: UpOscillantAxle -  An input signal is too low / Short circuit to ground";
  gc_ErrTranslation_fr_Text418 : WSTRING(84) := " [PIN_132 ]: UpOscillantAxle -  An input signal is too high / Short circuit to power";
  gc_ErrTranslation_fr_Text419 : WSTRING(69) := " [PIN_132 ]: UpOscillantAxle -  An input signal is out of valid range";
  gc_ErrTranslation_fr_Text420 : WSTRING(71) := " [PIN_132 ]: UpOscillantAxle -  Warning: a block has limited parameters";
  gc_ErrTranslation_fr_Text421 : WSTRING(55) := " [PIN_132 ]: UpOscillantAxle -  An initialization error";
  gc_ErrTranslation_fr_Text422 : WSTRING(79) := " [PIN_109 ]: UpFixeAxle -  An input signal is too low / Short circuit to ground";
  gc_ErrTranslation_fr_Text423 : WSTRING(79) := " [PIN_109 ]: UpFixeAxle -  An input signal is too high / Short circuit to power";
  gc_ErrTranslation_fr_Text424 : WSTRING(64) := " [PIN_109 ]: UpFixeAxle -  An input signal is out of valid range";
  gc_ErrTranslation_fr_Text425 : WSTRING(66) := " [PIN_109 ]: UpFixeAxle -  Warning: a block has limited parameters";
  gc_ErrTranslation_fr_Text426 : WSTRING(50) := " [PIN_109 ]: UpFixeAxle -  An initialization error";
  gc_ErrTranslation_fr_Text427 : WSTRING(73) := " [PIN_252 ]: PvgLeftTrackLowside -  HS OpenLoad / Short To Power external";
  gc_ErrTranslation_fr_Text428 : WSTRING(62) := " [PIN_252 ]: PvgLeftTrackLowside -  HS Short To Power internal";
  gc_ErrTranslation_fr_Text429 : WSTRING(54) := " [PIN_252 ]: PvgLeftTrackLowside -  HS Short To Ground";
  gc_ErrTranslation_fr_Text430 : WSTRING(57) := " [PIN_252 ]: PvgLeftTrackLowside -  Internal Driver Error";
  gc_ErrTranslation_fr_Text431 : WSTRING(27) := " [-]: SpecificErrorC1_2 -  ";
  gc_ErrTranslation_fr_Text432 : WSTRING(27) := " [-]: SpecificErrorC1_2 -  ";
  gc_ErrTranslation_fr_Text433 : WSTRING(27) := " [-]: SpecificErrorC1_2 -  ";
  gc_ErrTranslation_fr_Text434 : WSTRING(69) := " [-]: SpecificErrorC1_2 -  Inconsistency Nc No logical frame rotation";
  gc_ErrTranslation_fr_Text435 : WSTRING(27) := " [-]: SpecificErrorC1_2 -  ";
  gc_ErrTranslation_fr_Text436 : WSTRING(27) := " [-]: SpecificErrorC1_2 -  ";
  gc_ErrTranslation_fr_Text437 : WSTRING(85) := " [PIN_111 ]: FaultPvgDeltaArm -  An input signal is too low / Short circuit to ground";
  gc_ErrTranslation_fr_Text438 : WSTRING(85) := " [PIN_111 ]: FaultPvgDeltaArm -  An input signal is too high / Short circuit to power";
  gc_ErrTranslation_fr_Text439 : WSTRING(70) := " [PIN_111 ]: FaultPvgDeltaArm -  An input signal is out of valid range";
  gc_ErrTranslation_fr_Text440 : WSTRING(72) := " [PIN_111 ]: FaultPvgDeltaArm -  Warning: a block has limited parameters";
  gc_ErrTranslation_fr_Text441 : WSTRING(56) := " [PIN_111 ]: FaultPvgDeltaArm -  An initialization error";
  gc_ErrTranslation_fr_Text442 : WSTRING(85) := " [PIN_135 ]: FaultPvgArrowArm -  An input signal is too low / Short circuit to ground";
  gc_ErrTranslation_fr_Text443 : WSTRING(85) := " [PIN_135 ]: FaultPvgArrowArm -  An input signal is too high / Short circuit to power";
  gc_ErrTranslation_fr_Text444 : WSTRING(70) := " [PIN_135 ]: FaultPvgArrowArm -  An input signal is out of valid range";
  gc_ErrTranslation_fr_Text445 : WSTRING(72) := " [PIN_135 ]: FaultPvgArrowArm -  Warning: a block has limited parameters";
  gc_ErrTranslation_fr_Text446 : WSTRING(56) := " [PIN_135 ]: FaultPvgArrowArm -  An initialization error";
  gc_ErrTranslation_fr_Text447 : WSTRING(89) := " [PIN_112 ]: FaultPvgTelescopeArm -  An input signal is too low / Short circuit to ground";
  gc_ErrTranslation_fr_Text448 : WSTRING(89) := " [PIN_112 ]: FaultPvgTelescopeArm -  An input signal is too high / Short circuit to power";
  gc_ErrTranslation_fr_Text449 : WSTRING(74) := " [PIN_112 ]: FaultPvgTelescopeArm -  An input signal is out of valid range";
  gc_ErrTranslation_fr_Text450 : WSTRING(76) := " [PIN_112 ]: FaultPvgTelescopeArm -  Warning: a block has limited parameters";
  gc_ErrTranslation_fr_Text451 : WSTRING(60) := " [PIN_112 ]: FaultPvgTelescopeArm -  An initialization error";
  gc_ErrTranslation_fr_Text452 : WSTRING(85) := " [PIN_136 ]: FaultPvgEvProTOR -  An input signal is too low / Short circuit to ground";
  gc_ErrTranslation_fr_Text453 : WSTRING(85) := " [PIN_136 ]: FaultPvgEvProTOR -  An input signal is too high / Short circuit to power";
  gc_ErrTranslation_fr_Text454 : WSTRING(70) := " [PIN_136 ]: FaultPvgEvProTOR -  An input signal is out of valid range";
  gc_ErrTranslation_fr_Text455 : WSTRING(72) := " [PIN_136 ]: FaultPvgEvProTOR -  Warning: a block has limited parameters";
  gc_ErrTranslation_fr_Text456 : WSTRING(61) := " [PIN_161 ]: PvgLeftTrack -  Short to Power has been detected";
  gc_ErrTranslation_fr_Text457 : WSTRING(62) := " [PIN_161 ]: PvgLeftTrack -  Short to Ground has been detected";
  gc_ErrTranslation_fr_Text458 : WSTRING(44) := " [PIN_161 ]: PvgLeftTrack -  Wrong Parameter";
  gc_ErrTranslation_fr_Text459 : WSTRING(42) := " [PIN_161 ]: PvgLeftTrack -  Unknown error";
  gc_ErrTranslation_fr_Text460 : WSTRING(62) := " [PIN_185 ]: PvgRightTrack -  Short to Power has been detected";
  gc_ErrTranslation_fr_Text461 : WSTRING(63) := " [PIN_185 ]: PvgRightTrack -  Short to Ground has been detected";
  gc_ErrTranslation_fr_Text462 : WSTRING(45) := " [PIN_185 ]: PvgRightTrack -  Wrong Parameter";
  gc_ErrTranslation_fr_Text463 : WSTRING(43) := " [PIN_185 ]: PvgRightTrack -  Unknown error";
  gc_ErrTranslation_fr_Text464 : WSTRING(56) := " [PIN_136 ]: FaultPvgEvProTOR -  An initialization error";
  gc_ErrTranslation_fr_Text465 : WSTRING(32) := "Short to Power has been detected";
  gc_ErrTranslation_fr_Text466 : WSTRING(33) := "Short to Ground has been detected";
  gc_ErrTranslation_fr_Text467 : WSTRING(15) := "Wrong Parameter";
  gc_ErrTranslation_fr_Text468 : WSTRING(13) := "Unknown error";
  gc_ErrTranslation_fr_Text469 : WSTRING(37) := "HS OpenLoad / Short To Power external";
  gc_ErrTranslation_fr_Text470 : WSTRING(26) := "HS Short To Power internal";
  gc_ErrTranslation_fr_Text471 : WSTRING(18) := "HS Short To Ground";
  gc_ErrTranslation_fr_Text472 : WSTRING(21) := "Internal Driver Error";
  gc_ErrTranslation_fr_Text473 : WSTRING(37) := "HS OpenLoad / Short To Power external";
  gc_ErrTranslation_fr_Text474 : WSTRING(26) := "HS Short To Power internal";
  gc_ErrTranslation_fr_Text475 : WSTRING(71) := " [PIN_130 ]: BypassPressureSensor -  Master input signal short to power";
  gc_ErrTranslation_fr_Text476 : WSTRING(72) := " [PIN_130 ]: BypassPressureSensor -  Master input signal short to ground";
  gc_ErrTranslation_fr_Text477 : WSTRING(72) := " [PIN_130 ]: BypassPressureSensor -  Parameter of input char NOT monoton";
  gc_ErrTranslation_fr_Text478 : WSTRING(59) := " [PIN_130 ]: BypassPressureSensor -  Unknown internal error";
  gc_ErrTranslation_fr_Text479 : WSTRING(70) := " [PIN_108 PIN_146 ]: DownFixeAxle -  Logical Error between pin 0 and 1";
  gc_ErrTranslation_fr_Text480 : WSTRING(55) := " [PIN_108 PIN_146 ]: DownFixeAxle -  Vin0 < u16VolLoMin";
  gc_ErrTranslation_fr_Text481 : WSTRING(55) := " [PIN_108 PIN_146 ]: DownFixeAxle -  Vin0 > u16VolHiMax";
  gc_ErrTranslation_fr_Text482 : WSTRING(69) := " [PIN_108 PIN_146 ]: DownFixeAxle -  u16VolLoMax < Vin0 < u16VolHiMin";
  gc_ErrTranslation_fr_Text483 : WSTRING(55) := " [PIN_108 PIN_146 ]: DownFixeAxle -  Vin1 < u16VolLoMin";
  gc_ErrTranslation_fr_Text484 : WSTRING(55) := " [PIN_108 PIN_146 ]: DownFixeAxle -  Vin1 > u16VolHiMax";
  gc_ErrTranslation_fr_Text485 : WSTRING(69) := " [PIN_108 PIN_146 ]: DownFixeAxle -  u16VolLoMax < Vin1 < u16VolHiMin";
  gc_ErrTranslation_fr_Text486 : WSTRING(52) := "An input signal is too high / Short circuit to power";
  gc_ErrTranslation_fr_Text487 : WSTRING(37) := "An input signal is out of valid range";
  gc_ErrTranslation_fr_Text488 : WSTRING(52) := " [PIN_106 ]: GasGauge -  Input signal short to power";
  gc_ErrTranslation_fr_Text489 : WSTRING(53) := " [PIN_106 ]: GasGauge -  Input signal short to ground";
  gc_ErrTranslation_fr_Text490 : WSTRING(45) := " [PIN_106 ]: GasGauge -  Internal Block error";
  gc_ErrTranslation_fr_Text491 : WSTRING(39) := "Warning: a block has limited parameters";
  gc_ErrTranslation_fr_Text492 : WSTRING(23) := "An initialization error";
  gc_ErrTranslation_fr_Text493 : WSTRING(49) := "Openload detected on red light ARD output of 48xs";
  gc_ErrTranslation_fr_Text494 : WSTRING(33) := "Fault on thermic or electric pump";
  gc_ErrTranslation_fr_Text495 : WSTRING(11) := "Error bit 2";
  gc_ErrTranslation_fr_Text496 : WSTRING(11) := "Error bit 3";
  gc_ErrTranslation_fr_Text497 : WSTRING(11) := "Error bit 4";
  gc_ErrTranslation_fr_Text498 : WSTRING(11) := "Error bit 5";
  gc_ErrTranslation_fr_Text499 : WSTRING(74) := " [PIN_239 ]: PvgRightTrackLowside -  HS OpenLoad / Short To Power external";
  gc_ErrTranslation_fr_Text500 : WSTRING(63) := " [PIN_239 ]: PvgRightTrackLowside -  HS Short To Power internal";
  gc_ErrTranslation_fr_Text501 : WSTRING(55) := " [PIN_239 ]: PvgRightTrackLowside -  HS Short To Ground";
  gc_ErrTranslation_fr_Text502 : WSTRING(58) := " [PIN_239 ]: PvgRightTrackLowside -  Internal Driver Error";
  gc_ErrTranslation_fr_Text503 : WSTRING(78) := " [PIN_133 PIN_107 ]: FrameRotationSensor1 -  Logical Error between pin 0 and 1";
  gc_ErrTranslation_fr_Text504 : WSTRING(63) := " [PIN_133 PIN_107 ]: FrameRotationSensor1 -  Vin0 < u16VolLoMin";
  gc_ErrTranslation_fr_Text505 : WSTRING(63) := " [PIN_133 PIN_107 ]: FrameRotationSensor1 -  Vin0 > u16VolHiMax";
  gc_ErrTranslation_fr_Text506 : WSTRING(77) := " [PIN_133 PIN_107 ]: FrameRotationSensor1 -  u16VolLoMax < Vin0 < u16VolHiMin";
  gc_ErrTranslation_fr_Text507 : WSTRING(63) := " [PIN_133 PIN_107 ]: FrameRotationSensor1 -  Vin1 < u16VolLoMin";
  gc_ErrTranslation_fr_Text508 : WSTRING(63) := " [PIN_133 PIN_107 ]: FrameRotationSensor1 -  Vin1 > u16VolHiMax";
  gc_ErrTranslation_fr_Text509 : WSTRING(77) := " [PIN_133 PIN_107 ]: FrameRotationSensor1 -  u16VolLoMax < Vin1 < u16VolHiMin";
  gc_ErrTranslation_fr_Text510 : WSTRING(78) := " [PIN_114 PIN_112 ]: FrameRotationSensor2 -  Logical Error between pin 0 and 1";
  gc_ErrTranslation_fr_Text511 : WSTRING(63) := " [PIN_114 PIN_112 ]: FrameRotationSensor2 -  Vin0 < u16VolLoMin";
  gc_ErrTranslation_fr_Text512 : WSTRING(63) := " [PIN_114 PIN_112 ]: FrameRotationSensor2 -  Vin0 > u16VolHiMax";
  gc_ErrTranslation_fr_Text513 : WSTRING(77) := " [PIN_114 PIN_112 ]: FrameRotationSensor2 -  u16VolLoMax < Vin0 < u16VolHiMin";
  gc_ErrTranslation_fr_Text514 : WSTRING(63) := " [PIN_114 PIN_112 ]: FrameRotationSensor2 -  Vin1 < u16VolLoMin";
  gc_ErrTranslation_fr_Text515 : WSTRING(63) := " [PIN_114 PIN_112 ]: FrameRotationSensor2 -  Vin1 > u16VolHiMax";
  gc_ErrTranslation_fr_Text516 : WSTRING(77) := " [PIN_114 PIN_112 ]: FrameRotationSensor2 -  u16VolLoMax < Vin1 < u16VolHiMin";
  gc_ErrTranslation_fr_Text517 : WSTRING(11) := "Error bit 6";
  gc_ErrTranslation_fr_Text518 : WSTRING(11) := "Error bit 7";
  gc_ErrTranslation_fr_Text519 : WSTRING(52) := "An input signal is too low / Short circuit to ground";
  gc_ErrTranslation_fr_Text520 : WSTRING(52) := "An input signal is too high / Short circuit to power";
  gc_ErrTranslation_fr_Text521 : WSTRING(37) := "An input signal is out of valid range";
  gc_ErrTranslation_fr_Text522 : WSTRING(39) := "Warning: a block has limited parameters";
  gc_ErrTranslation_fr_Text523 : WSTRING(37) := "HS OpenLoad / Short To Power external";
  gc_ErrTranslation_fr_Text524 : WSTRING(26) := "HS Short To Power internal";
  gc_ErrTranslation_fr_Text525 : WSTRING(18) := "HS Short To Ground";
  gc_ErrTranslation_fr_Text526 : WSTRING(21) := "Internal Driver Error";
  gc_ErrTranslation_fr_Text527 : WSTRING(37) := "HS OpenLoad / Short To Power external";
  gc_ErrTranslation_fr_Text528 : WSTRING(26) := "HS Short To Power internal";
  gc_ErrTranslation_fr_Text529 : WSTRING(18) := "HS Short To Ground";
  gc_ErrTranslation_fr_Text530 : WSTRING(21) := "Internal Driver Error";
  gc_ErrTranslation_fr_Text531 : WSTRING(37) := "HS OpenLoad / Short To Power external";
  gc_ErrTranslation_fr_Text532 : WSTRING(26) := "HS Short To Power internal";
  gc_ErrTranslation_fr_Text533 : WSTRING(18) := "HS Short To Ground";
  gc_ErrTranslation_fr_Text534 : WSTRING(21) := "Internal Driver Error";
  gc_ErrTranslation_fr_Text535 : WSTRING(37) := "HS OpenLoad / Short To Power external";
  gc_ErrTranslation_fr_Text536 : WSTRING(26) := "HS Short To Power internal";
  gc_ErrTranslation_fr_Text537 : WSTRING(18) := "HS Short To Ground";
  gc_ErrTranslation_fr_Text538 : WSTRING(21) := "Internal Driver Error";
  gc_ErrTranslation_fr_Text539 : WSTRING(23) := "An initialization error";
  gc_ErrTranslation_fr_Text540 : WSTRING(34) := "Master input signal short to power";
  gc_ErrTranslation_fr_Text541 : WSTRING(35) := "Master input signal short to ground";
  gc_ErrTranslation_fr_Text542 : WSTRING(35) := "Parameter of input char NOT monoton";
  gc_ErrTranslation_fr_Text543 : WSTRING(22) := "Unknown internal error";
  gc_ErrTranslation_fr_Text544 : WSTRING(34) := "Master input signal short to power";
  gc_ErrTranslation_fr_Text545 : WSTRING(35) := "Master input signal short to ground";
  gc_ErrTranslation_fr_Text546 : WSTRING(35) := "Parameter of input char NOT monoton";
  gc_ErrTranslation_fr_Text547 : WSTRING(22) := "Unknown internal error";
  gc_ErrTranslation_fr_Text548 : WSTRING(18) := "HS Short To Ground";
  gc_ErrTranslation_fr_Text549 : WSTRING(21) := "Internal Driver Error";
  gc_ErrTranslation_fr_Text550 : WSTRING(37) := "HS OpenLoad / Short To Power external";
  gc_ErrTranslation_fr_Text551 : WSTRING(26) := "HS Short To Power internal";
  gc_ErrTranslation_fr_Text552 : WSTRING(18) := "HS Short To Ground";
  gc_ErrTranslation_fr_Text553 : WSTRING(21) := "Internal Driver Error";
  gc_ErrTranslation_fr_Text554 : WSTRING(37) := "HS OpenLoad / Short To Power external";
  gc_ErrTranslation_fr_Text555 : WSTRING(26) := "HS Short To Power internal";
  gc_ErrTranslation_fr_Text556 : WSTRING(18) := "HS Short To Ground";
  gc_ErrTranslation_fr_Text557 : WSTRING(21) := "Internal Driver Error";
  gc_ErrTranslation_fr_Text558 : WSTRING(80) := " [PIN_251 ]: ReturnLowSideEvForwardPump -  HS OpenLoad / Short To Power external";
  gc_ErrTranslation_fr_Text559 : WSTRING(69) := " [PIN_251 ]: ReturnLowSideEvForwardPump -  HS Short To Power internal";
  gc_ErrTranslation_fr_Text560 : WSTRING(61) := " [PIN_251 ]: ReturnLowSideEvForwardPump -  HS Short To Ground";
  gc_ErrTranslation_fr_Text561 : WSTRING(64) := " [PIN_251 ]: ReturnLowSideEvForwardPump -  Internal Driver Error";
  gc_ErrTranslation_fr_Text562 : WSTRING(81) := " [PIN_238 ]: ReturnLowSideEvBackwardPump -  HS OpenLoad / Short To Power external";
  gc_ErrTranslation_fr_Text563 : WSTRING(70) := " [PIN_238 ]: ReturnLowSideEvBackwardPump -  HS Short To Power internal";
  gc_ErrTranslation_fr_Text564 : WSTRING(62) := " [PIN_238 ]: ReturnLowSideEvBackwardPump -  HS Short To Ground";
  gc_ErrTranslation_fr_Text565 : WSTRING(37) := "HS OpenLoad / Short To Power external";
  gc_ErrTranslation_fr_Text566 : WSTRING(26) := "HS Short To Power internal";
  gc_ErrTranslation_fr_Text567 : WSTRING(18) := "HS Short To Ground";
  gc_ErrTranslation_fr_Text568 : WSTRING(21) := "Internal Driver Error";
  gc_ErrTranslation_fr_Text569 : WSTRING(37) := "HS OpenLoad / Short To Power external";
  gc_ErrTranslation_fr_Text570 : WSTRING(65) := " [PIN_238 ]: ReturnLowSideEvBackwardPump -  Internal Driver Error";
  gc_ErrTranslation_fr_Text571 : WSTRING(26) := "HS Short To Power internal";
  gc_ErrTranslation_fr_Text572 : WSTRING(18) := "HS Short To Ground";
  gc_ErrTranslation_fr_Text573 : WSTRING(21) := "Internal Driver Error";
  gc_ErrTranslation_fr_Text574 : WSTRING(32) := "Short to Power has been detected";
  gc_ErrTranslation_fr_Text575 : WSTRING(33) := "Short to Ground has been detected";
  gc_ErrTranslation_fr_Text576 : WSTRING(73) := " [PIN_177 ]: EvSelectorRotTurret -  HS OpenLoad / Short To Power external";
  gc_ErrTranslation_fr_Text577 : WSTRING(62) := " [PIN_177 ]: EvSelectorRotTurret -  HS Short To Power internal";
  gc_ErrTranslation_fr_Text578 : WSTRING(54) := " [PIN_177 ]: EvSelectorRotTurret -  HS Short To Ground";
  gc_ErrTranslation_fr_Text579 : WSTRING(57) := " [PIN_177 ]: EvSelectorRotTurret -  Internal Driver Error";
  gc_ErrTranslation_fr_Text580 : WSTRING(66) := " [PIN_163 ]: KlaxonNeotec -  HS OpenLoad / Short To Power external";
  gc_ErrTranslation_fr_Text581 : WSTRING(55) := " [PIN_163 ]: KlaxonNeotec -  HS Short To Power internal";
  gc_ErrTranslation_fr_Text582 : WSTRING(47) := " [PIN_163 ]: KlaxonNeotec -  HS Short To Ground";
  gc_ErrTranslation_fr_Text583 : WSTRING(50) := " [PIN_163 ]: KlaxonNeotec -  Internal Driver Error";
  gc_ErrTranslation_fr_Text584 : WSTRING(78) := " [PIN_177 ]: EvUnBlockOscillationAxle -  HS OpenLoad / Short To Power external";
  gc_ErrTranslation_fr_Text585 : WSTRING(79) := " [PIN_124 ]: ActiveHelp -  An input signal is too low / Short circuit to ground";
  gc_ErrTranslation_fr_Text586 : WSTRING(79) := " [PIN_124 ]: ActiveHelp -  An input signal is too high / Short circuit to power";
  gc_ErrTranslation_fr_Text587 : WSTRING(64) := " [PIN_124 ]: ActiveHelp -  An input signal is out of valid range";
  gc_ErrTranslation_fr_Text588 : WSTRING(66) := " [PIN_124 ]: ActiveHelp -  Warning: a block has limited parameters";
  gc_ErrTranslation_fr_Text589 : WSTRING(50) := " [PIN_124 ]: ActiveHelp -  An initialization error";
  gc_ErrTranslation_fr_Text590 : WSTRING(67) := " [PIN_177 ]: EvUnBlockOscillationAxle -  HS Short To Power internal";
  gc_ErrTranslation_fr_Text591 : WSTRING(59) := " [PIN_177 ]: EvUnBlockOscillationAxle -  HS Short To Ground";
  gc_ErrTranslation_fr_Text592 : WSTRING(62) := " [PIN_177 ]: EvUnBlockOscillationAxle -  Internal Driver Error";
  gc_ErrTranslation_fr_Text593 : WSTRING(78) := " [PIN_186 ]: EvParkBrakeAxleOscillant -  HS OpenLoad / Short To Power external";
  gc_ErrTranslation_fr_Text594 : WSTRING(67) := " [PIN_186 ]: EvParkBrakeAxleOscillant -  HS Short To Power internal";
  gc_ErrTranslation_fr_Text595 : WSTRING(59) := " [PIN_186 ]: EvParkBrakeAxleOscillant -  HS Short To Ground";
  gc_ErrTranslation_fr_Text596 : WSTRING(62) := " [PIN_186 ]: EvParkBrakeAxleOscillant -  Internal Driver Error";
  gc_ErrTranslation_fr_Text597 : WSTRING(73) := " [PIN_162 ]: EvParkBrakeAxleFixe -  HS OpenLoad / Short To Power external";
  gc_ErrTranslation_fr_Text598 : WSTRING(62) := " [PIN_162 ]: EvParkBrakeAxleFixe -  HS Short To Power internal";
  gc_ErrTranslation_fr_Text599 : WSTRING(54) := " [PIN_162 ]: EvParkBrakeAxleFixe -  HS Short To Ground";
  gc_ErrTranslation_fr_Text600 : WSTRING(57) := " [PIN_162 ]: EvParkBrakeAxleFixe -  Internal Driver Error";
  gc_ErrTranslation_fr_Text601 : WSTRING(81) := " [PIN_189 ]: EvServiceBrakeAxleOscillant -  HS OpenLoad / Short To Power external";
  gc_ErrTranslation_fr_Text602 : WSTRING(70) := " [PIN_189 ]: EvServiceBrakeAxleOscillant -  HS Short To Power internal";
  gc_ErrTranslation_fr_Text603 : WSTRING(62) := " [PIN_189 ]: EvServiceBrakeAxleOscillant -  HS Short To Ground";
  gc_ErrTranslation_fr_Text604 : WSTRING(15) := "Wrong Parameter";
  gc_ErrTranslation_fr_Text605 : WSTRING(13) := "Unknown error";
  gc_ErrTranslation_fr_Text606 : WSTRING(32) := "Short to Power has been detected";
  gc_ErrTranslation_fr_Text607 : WSTRING(33) := "Short to Ground has been detected";
  gc_ErrTranslation_fr_Text608 : WSTRING(15) := "Wrong Parameter";
  gc_ErrTranslation_fr_Text609 : WSTRING(56) := " [PIN_180 ]: EvPropGenerator -  Open load / open circuit";
  gc_ErrTranslation_fr_Text610 : WSTRING(71) := " [PIN_180 ]: EvPropGenerator -  Short circuit to power supply / battery";
  gc_ErrTranslation_fr_Text611 : WSTRING(55) := " [PIN_180 ]: EvPropGenerator -  Short circuit to ground";
